KUKA KRL program: MyProgram_153().src

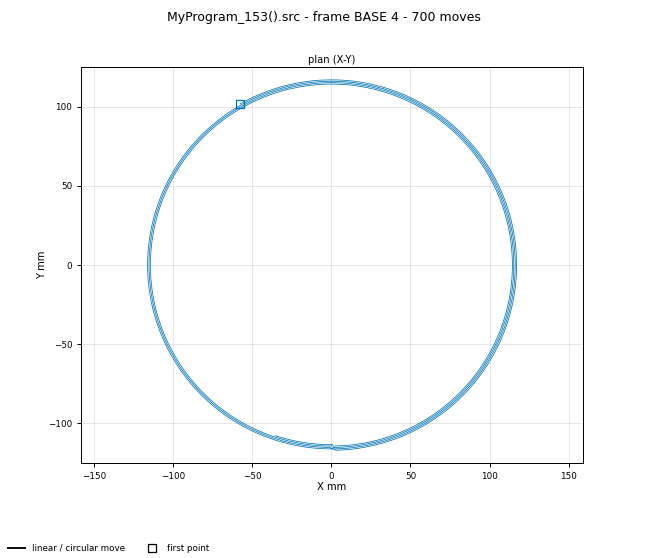
[picture p0: tool path of MyProgram_153().src in frame BASE 4, 700 of 700 moves have a stored position in this frame; points joined in program order, loops and branches not executed]
&ACCESS RVP
&REL 1
&PARAM TEMPLATE = C:\KRC\Roboter\Template\vorgabe
&PARAM EDITMASK = *
DEF MyProgram_153()
; ---- Setting reference (Base) ----
$BASE = BASE_DATA[4]

; --------------------------
; ---- Setting tool (TCP) ----
$TOOL = TOOL_DATA[3]
; --------------------------

$VEL.CP = VEL_APROX_PRINT
Startdeposition()
$VEL.CP = VEL_PRINT
LIN {X -57.7236,Y 101.8964,Z 119,A 114.9153,B 24.9392,C -1.8008,E1 24.9221,E2 331.1013} C_DIS
LIN {X -55.2055,Y 103.2823,Z 119,A 113.5039,B 24.9391,C -1.803,E1 24.9256,E2 332.5114} C_DIS
LIN {X -52.6542,Y 104.606,Z 119,A 112.0926,B 24.9389,C -1.8052,E1 24.9291,E2 333.9216} C_DIS
LIN {X -49.1645,Y 106.2888,Z 119,A 110.1729,B 24.9388,C -1.8071,E1 24.9339,E2 335.8414} C_DIS
LIN {X -46.1406,Y 107.638,Z 119,A 108.5652,B 24.9386,C -1.81,E1 24.938,E2 337.446} C_DIS
LIN {X -43.7577,Y 108.627,Z 119,A 107.2769,B 24.9386,C -1.8107,E1 24.9413,E2 338.7355} C_DIS
LIN {X -40.8035,Y 109.7723,Z 119,A 105.7445,B 24.9384,C -1.8135,E1 24.9453,E2 340.2645} C_DIS
LIN {X -38.3749,Y 110.6432,Z 119,A 104.5039,B 24.9382,C -1.8161,E1 24.9486,E2 341.5015} C_DIS
LIN {X -35.3681,Y 111.6422,Z 119,A 102.9247,B 24.9382,C -1.8167,E1 24.9528,E2 343.0821} C_DIS
LIN {X -32.8997,Y 112.3929,Z 119,A 101.6757,B 24.938,C -1.8187,E1 24.9561,E2 344.3285} C_DIS
LIN {X -30.1315,Y 113.1665,Z 119,A 100.2276,B 24.938,C -1.8184,E1 24.96,E2 345.7796} C_DIS
LIN {X -27.0594,Y 113.9416,Z 119,A 98.6962,B 24.9379,C -1.8206,E1 24.9642,E2 347.3077} C_DIS
LIN {X -24.5424,Y 114.5086,Z 119,A 97.4094,B 24.9379,C -1.8207,E1 24.9677,E2 348.5959} C_DIS
LIN {X -21.7248,Y 115.0764,Z 119,A 96.023,B 24.9377,C -1.8227,E1 24.9715,E2 349.979} C_DIS
LIN {X -18.8941,Y 115.5749,Z 119,A 94.5921,B 24.9377,C -1.8227,E1 24.9754,E2 351.4114} C_DIS
LIN {X -16.1821,Y 115.9853,Z 119,A 93.2548,B 24.9377,C -1.8238,E1 24.9791,E2 352.7472} C_DIS
LIN {X -12.9082,Y 116.397,Z 119,A 91.6544,B 24.9375,C -1.8253,E1 24.9835,E2 354.3452} C_DIS
LIN {X -10.0478,Y 116.6787,Z 119,A 90.2465,B 24.9375,C -1.8259,E1 24.9875,E2 355.7523} C_DIS
LIN {X -7.1813,Y 116.8902,Z 119,A 88.839,B 24.9375,C -1.8265,E1 24.9914,E2 357.159} C_DIS
LIN {X -4.3105,Y 117.0312,Z 119,A 87.4316,B 24.9375,C -1.8269,E1 24.9953,E2 358.5658} C_DIS
LIN {X -1.7313,Y 117.0963,Z 119,A 86.1688,B 24.9375,C -1.8272,E1 24.9988,E2 359.8279} C_DIS
LIN {X 1.4371,Y 117.1018,Z 119,A 84.6179,B 24.9375,C -1.8274,E1 25.0032,E2 361.3782} C_DIS
LIN {X 4.0165,Y 117.0403,Z 119,A 83.3552,B 24.9374,C -1.8276,E1 25.0067,E2 362.6403} C_DIS
LIN {X 7.1813,Y 116.8902,Z 119,A 81.8052,B 24.9374,C -1.8276,E1 25.011,E2 364.1896} C_DIS
LIN {X 10.0478,Y 116.6787,Z 119,A 80.399,B 24.9374,C -1.8275,E1 25.0149,E2 365.5954} C_DIS
LIN {X 12.9082,Y 116.397,Z 119,A 78.9934,B 24.9374,C -1.8273,E1 25.0188,E2 367.0004} C_DIS
LIN {X 15.7608,Y 116.0452,Z 119,A 77.5876,B 24.9374,C -1.827,E1 25.0227,E2 368.4058} C_DIS
LIN {X 18.3132,Y 115.6684,Z 119,A 76.3039,B 24.9375,C -1.8257,E1 25.0263,E2 369.6914} C_DIS
LIN {X 21.1464,Y 115.1841,Z 119,A 74.8988,B 24.9375,C -1.8252,E1 25.0301,E2 371.0961} C_DIS
LIN {X 23.9667,Y 114.6305,Z 119,A 73.4939,B 24.9375,C -1.8247,E1 25.034,E2 372.5007} C_DIS
LIN {X 26.7727,Y 114.0078,Z 119,A 72.1234,B 24.9375,C -1.8255,E1 25.0377,E2 373.8673} C_DIS
LIN {X 29.5625,Y 113.3164,Z 119,A 70.6849,B 24.9377,C -1.8232,E1 25.0416,E2 375.3091} C_DIS
LIN {X 32.3345,Y 112.5568,Z 119,A 69.2808,B 24.9377,C -1.8223,E1 25.0454,E2 376.7129} C_DIS
LIN {X 35.3681,Y 111.6422,Z 119,A 67.7553,B 24.9377,C -1.8223,E1 25.0494,E2 378.236} C_DIS
LIN {X 38.0973,Y 110.7406,Z 119,A 66.3515,B 24.9378,C -1.8211,E1 25.0531,E2 379.6396} C_DIS
LIN {X 40.5271,Y 109.8731,Z 119,A 65.0695,B 24.938,C -1.8191,E1 25.0565,E2 380.9237} C_DIS
LIN {X 43.2113,Y 108.8455,Z 119,A 63.6885,B 24.938,C -1.8188,E1 25.0601,E2 382.3024} C_DIS
LIN {X 45.7716,Y 107.7935,Z 119,A 62.3622,B 24.938,C -1.8186,E1 25.0635,E2 383.626} C_DIS
LIN {X 48.5001,Y 106.5941,Z 119,A 60.8826,B 24.9382,C -1.816,E1 25.0673,E2 385.1081} C_DIS
LIN {X 51.3666,Y 105.2443,Z 119,A 59.3365,B 24.9383,C -1.8142,E1 25.0712,E2 386.6544} C_DIS
LIN {X 53.672,Y 104.0859,Z 119,A 58.0778,B 24.9384,C -1.8128,E1 25.0743,E2 387.913} C_DIS
LIN {X 56.4688,Y 102.5971,Z 119,A 56.5322,B 24.9385,C -1.8108,E1 25.0781,E2 389.4588} C_DIS
LIN {X 58.9697,Y 101.1804,Z 119,A 55.1304,B 24.9387,C -1.809,E1 25.0815,E2 390.8608} C_DIS
LIN {X 61.435,Y 99.7027,Z 119,A 53.7287,B 24.9387,C -1.8071,E1 25.0849,E2 392.2626} C_DIS
LIN {X 63.8633,Y 98.165,Z 119,A 52.3274,B 24.9389,C -1.8051,E1 25.0881,E2 393.6641} C_DIS
LIN {X 67.1917,Y 95.9158,Z 119,A 50.3687,B 24.9391,C -1.8021,E1 25.0927,E2 395.6232} C_DIS
LIN {X 69.5253,Y 94.2379,Z 119,A 48.9459,B 24.9393,C -1.7989,E1 25.0959,E2 397.0486} C_DIS
LIN {X 72.0501,Y 92.3237,Z 119,A 47.424,B 24.9395,C -1.7973,E1 25.0992,E2 398.5686} C_DIS
LIN {X 74.2942,Y 90.5277,Z 119,A 46.023,B 24.9396,C -1.7949,E1 25.1023,E2 399.97} C_DIS
LIN {X 76.1743,Y 88.9491,Z 119,A 44.8121,B 24.9398,C -1.7921,E1 25.1049,E2 401.1827} C_DIS
LIN {X 78.6467,Y 86.7732,Z 119,A 43.2226,B 24.94,C -1.7899,E1 25.1082,E2 402.7713} C_DIS
LIN {X 80.5382,Y 85.0185,Z 119,A 41.9437,B 24.9402,C -1.7865,E1 25.1108,E2 404.0529} C_DIS
LIN {X 82.4233,Y 83.1914,Z 119,A 40.6216,B 24.9405,C -1.782,E1 25.1134,E2 405.3801} C_DIS
LIN {X 84.817,Y 80.7525,Z 119,A 39.0233,B 24.9405,C -1.7817,E1 25.1165,E2 406.9722} C_DIS
LIN {X 86.7732,Y 78.6467,Z 119,A 37.6237,B 24.9407,C -1.7788,E1 25.1192,E2 408.3724} C_DIS
LIN {X 89.4184,Y 75.6234,Z 119,A 35.6681,B 24.941,C -1.7747,E1 25.1227,E2 410.3289} C_DIS
LIN {X 91.2474,Y 73.4062,Z 119,A 34.2691,B 24.9412,C -1.7717,E1 25.1252,E2 411.7284} C_DIS
LIN {X 93.2009,Y 70.9117,Z 119,A 32.7271,B 24.9414,C -1.7683,E1 25.1278,E2 413.2713} C_DIS
LIN {X 95.424,Y 67.8871,Z 119,A 30.862,B 24.9418,C -1.7623,E1 25.1309,E2 415.1414} C_DIS
LIN {X 97.2089,Y 65.3068,Z 119,A 29.3517,B 24.942,C -1.7595,E1 25.1333,E2 416.6509} C_DIS
LIN {X 98.7132,Y 63.0092,Z 119,A 28.0222,B 24.9422,C -1.7567,E1 25.1353,E2 417.9804} C_DIS
LIN {X 100.2963,Y 60.4583,Z 119,A 26.5548,B 24.9424,C -1.7528,E1 25.1374,E2 419.4494} C_DIS
LIN {X 101.8964,Y 57.7236,Z 119,A 25.036,B 24.9426,C -1.75,E1 25.1396,E2 420.967} C_DIS
LIN {X 103.142,Y 55.4641,Z 119,A 23.7809,B 24.9428,C -1.7469,E1 25.1412,E2 422.2228} C_DIS
LIN {X 104.606,Y 52.6542,Z 119,A 22.2401,B 24.9431,C -1.743,E1 25.1432,E2 423.7647} C_DIS
LIN {X 105.7393,Y 50.3364,Z 119,A 20.9634,B 24.9433,C -1.7387,E1 25.1448,E2 425.0446} C_DIS
LIN {X 107.0636,Y 47.458,Z 119,A 19.4448,B 24.9435,C -1.7357,E1 25.1465,E2 426.5621} C_DIS
LIN {X 108.627,Y 43.7577,Z 119,A 17.4694,B 24.9439,C -1.7295,E1 25.1486,E2 428.5412} C_DIS
LIN {X 109.7723,Y 40.8035,Z 119,A 15.9513,B 24.9441,C -1.7264,E1 25.1501,E2 430.0582} C_DIS
LIN {X 110.6432,Y 38.3749,Z 119,A 14.6749,B 24.9444,C -1.722,E1 25.1513,E2 431.3379} C_DIS
LIN {X 111.5517,Y 35.648,Z 119,A 13.2998,B 24.9446,C -1.7192,E1 25.1525,E2 432.7118} C_DIS
LIN {X 112.3929,Y 32.8996,Z 119,A 11.9026,B 24.9449,C -1.7153,E1 25.1536,E2 434.1101} C_DIS
LIN {X 113.1665,Y 30.1315,Z 119,A 10.5341,B 24.945,C -1.7128,E1 25.1546,E2 435.4768} C_DIS
LIN {X 113.8718,Y 27.3452,Z 119,A 9.1088,B 24.9454,C -1.7075,E1 25.1556,E2 436.9064} C_DIS
LIN {X 114.5713,Y 24.2549,Z 119,A 7.5688,B 24.9456,C -1.7031,E1 25.1565,E2 438.4478} C_DIS
LIN {X 115.0764,Y 21.7248,Z 119,A 6.3152,B 24.9459,C -1.6995,E1 25.1572,E2 439.7024} C_DIS
LIN {X 115.5684,Y 18.9331,Z 119,A 4.9099,B 24.9462,C -1.6942,E1 25.1579,E2 441.1119} C_DIS
LIN {X 116.0038,Y 16.0521,Z 119,A 3.5219,B 24.9464,C -1.6915,E1 25.1584,E2 442.4983} C_DIS
LIN {X 116.397,Y 12.9082,Z 119,A 1.9824,B 24.9467,C -1.687,E1 25.1589,E2 444.0393} C_DIS
LIN {X 116.6517,Y 10.3407,Z 119,A 0.7286,B 24.9469,C -1.6833,E1 25.1592,E2 445.2942} C_DIS
LIN {X 116.8902,Y 7.1813,Z 119,A -0.8108,B 24.9472,C -1.6788,E1 25.1595,E2 446.8353} C_DIS
LIN {X 117.0312,Y 4.3105,Z 119,A -2.2075,B 24.9474,C -1.6747,E1 25.1597,E2 448.2333} C_DIS
LIN {X 117.0963,Y 1.7313,Z 119,A -3.497,B 24.9478,C -1.6693,E1 25.1597,E2 449.5278} C_DIS
LIN {X 117.0963,Y -1.7313,Z 119,A -5.014,B 24.9476,C -1.6722,E1 25.1597,E2 451.0289} C_DIS
LIN {X 117.0465,Y -3.8126,Z 119,A -6.1822,B 24.9483,C -1.6618,E1 25.1597,E2 452.2148} C_DIS
LIN {X 116.91,Y -6.8222,Z 119,A -7.6255,B 24.9485,C -1.6584,E1 25.1595,E2 453.6574} C_DIS
LIN {X 116.693,Y -9.8691,Z 119,A -9.1115,B 24.9487,C -1.6539,E1 25.1591,E2 455.1452} C_DIS
LIN {X 116.397,Y -12.9082,Z 119,A -10.586,B 24.949,C -1.6499,E1 25.1587,E2 456.6204} C_DIS
LIN {X 116.0452,Y -15.7608,Z 119,A -11.9826,B 24.9492,C -1.6458,E1 25.1582,E2 458.0185} C_DIS
LIN {X 115.6684,Y -18.3132,Z 119,A -13.2584,B 24.9495,C -1.6411,E1 25.1577,E2 459.2978} C_DIS
LIN {X 115.1321,Y -21.4359,Z 119,A -14.7758,B 24.9497,C -1.6376,E1 25.1569,E2 460.8147} C_DIS
LIN {X 114.6305,Y -23.9667,Z 119,A -16.0514,B 24.95,C -1.6329,E1 25.1562,E2 462.0939} C_DIS
LIN {X 114.0078,Y -26.7727,Z 119,A -17.426,B 24.9502,C -1.6299,E1 25.1554,E2 463.4677} C_DIS
LIN {X 113.3164,Y -29.5625,Z 119,A -18.8446,B 24.9505,C -1.6248,E1 25.1544,E2 464.89} C_DIS
LIN {X 112.2191,Y -33.4857,Z 119,A -20.8654,B 24.951,C -1.6171,E1 25.1528,E2 466.9174} C_DIS
LIN {X 111.2904,Y -36.4555,Z 119,A -22.3142,B 24.951,C -1.6157,E1 25.1516,E2 468.3612} C_DIS
LIN {X 110.4329,Y -38.9742,Z 119,A -23.6361,B 24.9514,C -1.6107,E1 25.1504,E2 469.6876} C_DIS
LIN {X 109.3675,Y -41.8724,Z 119,A -25.108,B 24.9516,C -1.6078,E1 25.1489,E2 471.158} C_DIS
LIN {X 108.1961,Y -44.8163,Z 119,A -26.6478,B 24.9518,C -1.6035,E1 25.1473,E2 472.6996} C_DIS
LIN {X 107.1812,Y -47.1884,Z 119,A -27.9239,B 24.9521,C -1.5989,E1 25.1459,E2 473.9794} C_DIS
LIN {X 105.8667,Y -50.0712,Z 119,A -29.442,B 24.9523,C -1.5957,E1 25.1441,E2 475.4969} C_DIS
LIN {X 104.606,Y -52.6542,Z 119,A -30.8392,B 24.9525,C -1.5919,E1 25.1424,E2 476.8956} C_DIS
LIN {X 103.4194,Y -54.9452,Z 119,A -32.0936,B 24.9527,C -1.5885,E1 25.1408,E2 478.1514} C_DIS
LIN {X 102.0398,Y -57.4667,Z 119,A -33.491,B 24.9529,C -1.5848,E1 25.1389,E2 479.5502} C_DIS
LIN {X 100.5988,Y -59.9536,Z 119,A -34.9105,B 24.9532,C -1.58,E1 25.1368,E2 480.9736} C_DIS
LIN {X 98.9413,Y -62.6539,Z 119,A -36.4291,B 24.9534,C -1.577,E1 25.1346,E2 482.4916} C_DIS
LIN {X 97.3739,Y -65.0632,Z 119,A -37.8269,B 24.9536,C -1.5734,E1 25.1325,E2 483.891} C_DIS
LIN {X 95.9158,Y -67.1917,Z 119,A -39.0816,B 24.9538,C -1.5703,E1 25.1305,E2 485.1469} C_DIS
LIN {X 94.352,Y -69.3694,Z 119,A -40.4109,B 24.9541,C -1.5658,E1 25.1283,E2 486.4804} C_DIS
LIN {X 92.5033,Y -71.8171,Z 119,A -41.8777,B 24.9542,C -1.5633,E1 25.1258,E2 487.9461} C_DIS
LIN {X 90.5277,Y -74.2942,Z 119,A -43.4188,B 24.9544,C -1.5595,E1 25.1231,E2 489.4889} C_DIS
LIN {X 88.868,Y -76.2695,Z 119,A -44.6741,B 24.9546,C -1.5566,E1 25.1208,E2 490.7455} C_DIS
LIN {X 86.7732,Y -78.6467,Z 119,A -46.2156,B 24.9548,C -1.5529,E1 25.1179,E2 492.2887} C_DIS
LIN {X 84.9044,Y -80.6596,Z 119,A -47.557,B 24.955,C -1.5497,E1 25.1154,E2 493.6319} C_DIS
LIN {X 82.8097,Y -82.8097,Z 119,A -49.0132,B 24.9552,C -1.5466,E1 25.1125,E2 495.0892} C_DIS
LIN {X 80.9643,Y -84.6128,Z 119,A -50.2689,B 24.9553,C -1.5439,E1 25.11,E2 496.3461} C_DIS
LIN {X 78.8634,Y -86.5743,Z 119,A -51.668,B 24.9555,C -1.5409,E1 25.1071,E2 497.7467} C_DIS
LIN {X 76.4935,Y -88.6772,Z 119,A -53.2105,B 24.9557,C -1.5376,E1 25.1039,E2 499.2907} C_DIS
LIN {X 74.5204,Y -90.3397,Z 119,A -54.467,B 24.9559,C -1.535,E1 25.1012,E2 500.5485} C_DIS
LIN {X 72.0501,Y -92.3237,Z 119,A -56.0095,B 24.956,C -1.5319,E1 25.0978,E2 502.0925} C_DIS
LIN {X 69.7627,Y -94.0641,Z 119,A -57.4095,B 24.9562,C -1.5292,E1 25.0947,E2 503.4938} C_DIS
LIN {X 67.4332,Y -95.7478,Z 119,A -58.8096,B 24.9563,C -1.5266,E1 25.0915,E2 504.8953} C_DIS
LIN {X 65.3068,Y -97.2089,Z 119,A -60.0666,B 24.9565,C -1.5243,E1 25.0886,E2 506.1534} C_DIS
LIN {X 62.9015,Y -98.7824,Z 119,A -61.4668,B 24.9566,C -1.5218,E1 25.0853,E2 507.555} C_DIS
LIN {X 60.4583,Y -100.2963,Z 119,A -62.8848,B 24.9568,C -1.5186,E1 25.0819,E2 508.9761} C_DIS
LIN {X 57.7236,Y -101.8964,Z 119,A -64.4114,B 24.9568,C -1.5168,E1 25.0782,E2 510.5023} C_DIS
LIN {X 55.2055,Y -103.2823,Z 119,A -65.8123,B 24.957,C -1.5146,E1 25.0748,E2 511.9044} C_DIS
LIN {X 52.884,Y -104.4886,Z 119,A -67.0847,B 24.9571,C -1.5128,E1 25.0716,E2 513.1776} C_DIS
LIN {X 50.3364,Y -105.7393,Z 119,A -68.4714,B 24.9572,C -1.5106,E1 25.0681,E2 514.5657} C_DIS
LIN {X 47.7263,Y -106.9428,Z 119,A -69.8951,B 24.9574,C -1.5076,E1 25.0645,E2 515.993} C_DIS
LIN {X 45.0874,Y -108.0818,Z 119,A -71.2747,B 24.9574,C -1.5068,E1 25.0609,E2 517.3714} C_DIS
LIN {X 42.1475,Y -109.2633,Z 119,A -72.8202,B 24.9576,C -1.5048,E1 25.0569,E2 518.9181} C_DIS
LIN {X 39.4534,Y -110.2648,Z 119,A -74.2224,B 24.9576,C -1.5031,E1 25.0532,E2 520.3214} C_DIS
LIN {X 36.7355,Y -111.1998,Z 119,A -75.6249,B 24.9578,C -1.5015,E1 25.0495,E2 521.725} C_DIS
LIN {X 34.2764,Y -111.9807,Z 119,A -76.8841,B 24.9578,C -1.5001,E1 25.0462,E2 522.9851} C_DIS
LIN {X 31.5179,Y -112.7882,Z 119,A -78.2869,B 24.9579,C -1.4987,E1 25.0424,E2 524.3888} C_DIS
LIN {X 28.4555,Y -113.6009,Z 119,A -79.8337,B 24.958,C -1.4972,E1 25.0382,E2 525.9368} C_DIS
LIN {X 26.1295,Y -114.1564,Z 119,A -81.026,B 24.9581,C -1.4951,E1 25.035,E2 527.1324} C_DIS
LIN {X 22.8471,Y -114.8603,Z 119,A -82.6405,B 24.9581,C -1.4949,E1 25.0306,E2 528.7455} C_DIS
LIN {X 20.311,Y -115.3344,Z 119,A -83.9008,B 24.9581,C -1.494,E1 25.0271,E2 530.0065} C_DIS
LIN {X 17.1837,Y -115.843,Z 119,A -85.4485,B 24.9582,C -1.4929,E1 25.0228,E2 531.5551} C_DIS
LIN {X 14.6273,Y -116.1921,Z 119,A -86.7314,B 24.9583,C -1.4912,E1 25.0193,E2 532.8411} C_DIS
LIN {X 11.7714,Y -116.516,Z 119,A -88.1136,B 24.9583,C -1.4915,E1 25.0154,E2 534.2218} C_DIS
LIN {X 8.9085,Y -116.7698,Z 119,A -89.5405,B 24.9584,C -1.4898,E1 25.0114,E2 535.6518} C_DIS
LIN {X 6.0401,Y -116.9533,Z 119,A -90.9095,B 24.9584,C -1.4909,E1 25.0076,E2 537.0177} C_DIS
LIN {X 2.874,Y -117.0753,Z 119,A -92.4722,B 24.9584,C -1.4898,E1 25.0033,E2 538.5827} C_DIS
LIN {X 2.874,Y -117.0753,Z 119,A -92.4722,B 24.9584,C -1.4898,E1 25.0033,E2 538.5827} C_DIS
Enddeposition()
LIN {X 0.8107,Y -116.2129,Z 119,A -92.8235,B 24.9559,C -1.5347,E1 25.0026,E2 538.8274} C_DIS
Startdeposition()
$VEL.CP = VEL_PRINT
LIN {X 4.253,Y -116.1409,Z 119,A -90.9838,B 24.9555,C -1.5417,E1 25.0078,E2 536.9717} C_DIS
LIN {X 8.3855,Y -115.9152,Z 119,A -89.0694,B 24.9557,C -1.5369,E1 25.0131,E2 535.0695} C_DIS
LIN {X 11.4655,Y -115.6516,Z 119,A -87.6523,B 24.956,C -1.5328,E1 25.017,E2 533.6628} C_DIS
LIN {X 14.4704,Y -115.3134,Z 119,A -85.9882,B 24.9555,C -1.5417,E1 25.0216,E2 531.979} C_DIS
LIN {X 18.8822,Y -114.673,Z 119,A -83.5014,B 24.9546,C -1.5565,E1 25.0286,E2 529.4595} C_DIS
LIN {X 22.2001,Y -114.077,Z 119,A -81.8222,B 24.9545,C -1.5587,E1 25.0332,E2 527.777} C_DIS
LIN {X 25.6561,Y -113.3507,Z 119,A -80.4241,B 24.9553,C -1.5446,E1 25.0369,E2 526.4143} C_DIS
LIN {X 30.8978,Y -112.0359,Z 119,A -77.7136,B 24.955,C -1.5494,E1 25.0443,E2 523.6965} C_DIS
LIN {X 34.2636,Y -111.0512,Z 119,A -76.0256,B 24.955,C -1.5496,E1 25.0488,E2 522.011} C_DIS
LIN {X 37.4676,Y -110.0121,Z 119,A -74.4944,B 24.9552,C -1.5457,E1 25.0528,E2 520.492} C_DIS
LIN {X 40.0272,Y -109.1065,Z 119,A -73.0582,B 24.9549,C -1.552,E1 25.0566,E2 519.0439} C_DIS
LIN {X 44.6117,Y -107.3148,Z 119,A -70.7821,B 24.9551,C -1.5485,E1 25.0625,E2 516.7813} C_DIS
LIN {X 47.9397,Y -105.8687,Z 119,A -68.956,B 24.9548,C -1.5529,E1 25.0671,E2 514.9491} C_DIS
LIN {X 51.1277,Y -104.3676,Z 119,A -66.9334,B 24.9539,C -1.569,E1 25.0723,E2 512.8938} C_DIS
LIN {X 55.4285,Y -102.1471,Z 119,A -64.8466,B 24.9545,C -1.5592,E1 25.0774,E2 510.8361} C_DIS
LIN {X 58.5784,Y -100.376,Z 119,A -63.1081,B 24.9544,C -1.5604,E1 25.0816,E2 509.1} C_DIS
LIN {X 60.8412,Y -99.0203,Z 119,A -61.7959,B 24.9542,C -1.5634,E1 25.0847,E2 507.7848} C_DIS
LIN {X 62.8687,Y -97.744,Z 119,A -60.6023,B 24.954,C -1.5663,E1 25.0876,E2 506.5882} C_DIS
LIN {X 65.3722,Y -96.0879,Z 119,A -59.0534,B 24.9537,C -1.5725,E1 25.0912,E2 505.0298} C_DIS
LIN {X 68.06,Y -94.2054,Z 119,A -57.5231,B 24.9537,C -1.5717,E1 25.0946,E2 503.5066} C_DIS
LIN {X 70.0238,Y -92.7529,Z 119,A -56.3173,B 24.9536,C -1.5744,E1 25.0973,E2 502.2989} C_DIS
LIN {X 72.184,Y -91.0815,Z 119,A -54.9676,B 24.9534,C -1.5775,E1 25.1003,E2 500.9468} C_DIS
LIN {X 74.9817,Y -88.7938,Z 119,A -53.1012,B 24.9529,C -1.5855,E1 25.1043,E2 499.0687} C_DIS
LIN {X 77.5595,Y -86.5499,Z 119,A -51.4398,B 24.9527,C -1.5884,E1 25.1078,E2 497.4072} C_DIS
LIN {X 79.9992,Y -84.3015,Z 119,A -49.914,B 24.9528,C -1.5871,E1 25.1109,E2 495.8907} C_DIS
LIN {X 81.9579,Y -82.3979,Z 119,A -48.4044,B 24.9521,C -1.5981,E1 25.1139,E2 494.3614} C_DIS
LIN {X 84.5156,Y -79.7716,Z 119,A -46.7091,B 24.9521,C -1.5973,E1 25.1172,E2 492.6753} C_DIS
LIN {X 87.0213,Y -77.0329,Z 119,A -44.7713,B 24.9516,C -1.6071,E1 25.1208,E2 490.7229} C_DIS
LIN {X 89.4873,Y -74.1512,Z 119,A -43.0863,B 24.9518,C -1.6033,E1 25.1238,E2 489.0547} C_DIS
LIN {X 91.1471,Y -72.101,Z 119,A -41.76,B 24.9515,C -1.608,E1 25.1262,E2 487.7234} C_DIS
LIN {X 93.2609,Y -69.3475,Z 119,A -40.0948,B 24.9515,C -1.6105,E1 25.129,E2 486.0604} C_DIS
LIN {X 95.3441,Y -66.452,Z 119,A -38.2246,B 24.9508,C -1.6207,E1 25.132,E2 484.175} C_DIS
LIN {X 97.3147,Y -63.5332,Z 119,A -36.3931,B 24.9502,C -1.6302,E1 25.1348,E2 482.3303} C_DIS
LIN {X 100.5499,Y -58.2774,Z 119,A -33.6602,B 24.9506,C -1.6242,E1 25.1388,E2 479.6255} C_DIS
LIN {X 101.9362,Y -55.8173,Z 119,A -32.1145,B 24.9499,C -1.6357,E1 25.1409,E2 478.0608} C_DIS
LIN {X 103.6714,Y -52.524,Z 119,A -29.9709,B 24.9486,C -1.656,E1 25.1436,E2 475.8807} C_DIS
LIN {X 105.143,Y -49.5133,Z 119,A -28.8351,B 24.9498,C -1.6362,E1 25.145,E2 474.7976} C_DIS
LIN {X 106.0516,Y -47.5339,Z 119,A -27.6856,B 24.9494,C -1.6432,E1 25.1463,E2 473.6381} C_DIS
LIN {X 107.4428,Y -44.3021,Z 119,A -26.0414,B 24.9494,C -1.6442,E1 25.1481,E2 472.0004} C_DIS
LIN {X 108.4294,Y -41.8321,Z 119,A -24.6571,B 24.9489,C -1.6518,E1 25.1495,E2 470.606} C_DIS
LIN {X 109.2722,Y -39.5727,Z 119,A -23.4046,B 24.9485,C -1.6586,E1 25.1507,E2 469.3445} C_DIS
LIN {X 110.5377,Y -35.8857,Z 119,A -21.4658,B 24.948,C -1.6655,E1 25.1524,E2 467.4004} C_DIS
LIN {X 111.4364,Y -32.9893,Z 119,A -20.0248,B 24.9479,C -1.6676,E1 25.1536,E2 465.9625} C_DIS
LIN {X 112.4888,Y -29.201,Z 119,A -18.0887,B 24.9475,C -1.6737,E1 25.155,E2 464.0231} C_DIS
LIN {X 113.4181,Y -25.3586,Z 119,A -16.0726,B 24.9469,C -1.6832,E1 25.1563,E2 461.9963} C_DIS
LIN {X 114.2163,Y -21.4768,Z 119,A -14.1057,B 24.9465,C -1.6902,E1 25.1573,E2 460.0245} C_DIS
LIN {X 114.9223,Y -17.3041,Z 119,A -12.1735,B 24.9465,C -1.6896,E1 25.1582,E2 458.1051} C_DIS
LIN {X 115.4268,Y -13.5277,Z 119,A -10.266,B 24.946,C -1.6971,E1 25.1588,E2 456.1911} C_DIS
LIN {X 115.7339,Y -10.5844,Z 119,A -8.8175,B 24.9458,C -1.7014,E1 25.1592,E2 454.7411} C_DIS
LIN {X 116.0065,Y -7.0137,Z 119,A -6.9886,B 24.9452,C -1.7102,E1 25.1596,E2 452.9024} C_DIS
LIN {X 116.1771,Y -3.0757,Z 119,A -5.2194,B 24.9453,C -1.7081,E1 25.1598,E2 451.1484} C_DIS
LIN {X 116.215,Y -0.6787,Z 119,A -4.0416,B 24.9451,C -1.7118,E1 25.1598,E2 449.9689} C_DIS
LIN {X 116.1972,Y 2.1365,Z 119,A -2.5867,B 24.9446,C -1.7196,E1 25.1598,E2 448.5045} C_DIS
LIN {X 116.1033,Y 5.1384,Z 119,A -1.1929,B 24.9446,C -1.7202,E1 25.1596,E2 447.1174} C_DIS
LIN {X 115.9024,Y 8.571,Z 119,A 0.4861,B 24.9442,C -1.7249,E1 25.1593,E2 445.4374} C_DIS
LIN {X 115.6815,Y 11.1514,Z 119,A 1.738,B 24.9441,C -1.7278,E1 25.159,E2 444.186} C_DIS
LIN {X 115.354,Y 14.1499,Z 119,A 3.2576,B 24.9436,C -1.7341,E1 25.1585,E2 442.6604} C_DIS
LIN {X 114.8631,Y 17.6866,Z 119,A 4.9746,B 24.9434,C -1.7377,E1 25.1578,E2 440.9451} C_DIS
LIN {X 114.3714,Y 20.6285,Z 119,A 6.5239,B 24.9429,C -1.7462,E1 25.157,E2 439.385} C_DIS
LIN {X 112.7269,Y 28.2747,Z 119,A 10.9009,B 24.9404,C -1.7832,E1 25.1543,E2 434.9462} C_DIS
LIN {X 111.6203,Y 32.3693,Z 119,A 12.3577,B 24.942,C -1.7592,E1 25.1532,E2 433.5542} C_DIS
LIN {X 110.8416,Y 34.9399,Z 119,A 13.8569,B 24.9412,C -1.7716,E1 25.1519,E2 432.0343} C_DIS
LIN {X 109.644,Y 38.5298,Z 119,A 15.5806,B 24.9412,C -1.7705,E1 25.1504,E2 430.323} C_DIS
LIN {X 108.5425,Y 41.5336,Z 119,A 17.2672,B 24.9406,C -1.7803,E1 25.1487,E2 428.6225} C_DIS
LIN {X 107.103,Y 45.1142,Z 119,A 18.9913,B 24.9408,C -1.7774,E1 25.1469,E2 426.9147} C_DIS
LIN {X 105.6303,Y 48.4665,Z 119,A 20.7455,B 24.9406,C -1.7802,E1 25.1449,E2 425.1635} C_DIS
LIN {X 104.2221,Y 51.4214,Z 119,A 22.4929,B 24.9399,C -1.7912,E1 25.1428,E2 423.3997} C_DIS
LIN {X 102.6122,Y 54.5646,Z 119,A 24.2036,B 24.9396,C -1.7946,E1 25.1405,E2 421.69} C_DIS
LIN {X 100.7406,Y 57.9455,Z 119,A 26.1314,B 24.9392,C -1.8009,E1 25.1379,E2 419.7574} C_DIS
LIN {X 98.8898,Y 61.0535,Z 119,A 27.8696,B 24.939,C -1.8035,E1 25.1354,E2 418.0219} C_DIS
LIN {X 96.4195,Y 64.8826,Z 119,A 30.1003,B 24.9387,C -1.8086,E1 25.132,E2 415.7901} C_DIS
LIN {X 94.333,Y 67.8812,Z 119,A 31.8188,B 24.9387,C -1.8093,E1 25.1292,E2 414.0784} C_DIS
LIN {X 92.5913,Y 70.2388,Z 119,A 33.5412,B 24.9375,C -1.8259,E1 25.1262,E2 412.325} C_DIS
LIN {X 90.3004,Y 73.1586,Z 119,A 35.1466,B 24.9379,C -1.8198,E1 25.1235,E2 410.7416} C_DIS
LIN {X 87.7708,Y 76.1759,Z 119,A 37.1508,B 24.9374,C -1.8273,E1 25.1198,E2 408.7288} C_DIS
LIN {X 84.9502,Y 79.3094,Z 119,A 38.9364,B 24.938,C -1.8183,E1 25.1165,E2 406.9722} C_DIS
LIN {X 83.3255,Y 81.0152,Z 119,A 40.2225,B 24.9375,C -1.8267,E1 25.114,E2 405.672} C_DIS
LIN {X 81.3391,Y 83.0092,Z 119,A 41.9399,B 24.9362,C -1.845,E1 25.1105,E2 403.9184} C_DIS
LIN {X 78.4661,Y 85.7289,Z 119,A 43.5948,B 24.9369,C -1.8353,E1 25.1072,E2 402.2932} C_DIS
LIN {X 75.7231,Y 88.1622,Z 119,A 45.5314,B 24.9362,C -1.8449,E1 25.1031,E2 400.3417} C_DIS
LIN {X 72.1095,Y 91.1404,Z 119,A 47.7484,B 24.9362,C -1.845,E1 25.0983,E2 398.1326} C_DIS
LIN {X 68.9027,Y 93.5888,Z 119,A 50.173,B 24.9345,C -1.8687,E1 25.0927,E2 395.6607} C_DIS
LIN {X 65.6694,Y 95.8867,Z 119,A 51.764,B 24.9355,C -1.8551,E1 25.0892,E2 394.1074} C_DIS
LIN {X 62.1674,Y 98.1939,Z 119,A 53.6266,B 24.9359,C -1.849,E1 25.0849,E2 392.2652} C_DIS
LIN {X 59.197,Y 100.0103,Z 119,A 55.4249,B 24.9355,C -1.8554,E1 25.0805,E2 390.4575} C_DIS
LIN {X 55.9099,Y 101.886,Z 119,A 57.1397,B 24.9358,C -1.8511,E1 25.0764,E2 388.7578} C_DIS
LIN {X 53.8271,Y 103.0007,Z 119,A 58.6381,B 24.9346,C -1.8679,E1 25.0726,E2 387.224} C_DIS
LIN {X 49.8879,Y 104.9657,Z 119,A 60.56,B 24.9352,C -1.8593,E1 25.0678,E2 385.3275} C_DIS
LIN {X 47.3698,Y 106.1255,Z 119,A 61.9307,B 24.9351,C -1.8611,E1 25.0643,E2 383.9561} C_DIS
LIN {X 44.1416,Y 107.5081,Z 119,A 63.7304,B 24.9347,C -1.866,E1 25.0597,E2 382.1488} C_DIS
LIN {X 41.5455,Y 108.538,Z 119,A 64.9955,B 24.935,C -1.8623,E1 25.0564,E2 380.8952} C_DIS
LIN {X 38.3682,Y 109.7007,Z 119,A 66.7171,B 24.9347,C -1.8663,E1 25.0519,E2 379.1678} C_DIS
LIN {X 35.2519,Y 110.7428,Z 119,A 68.2686,B 24.9348,C -1.8645,E1 25.0478,E2 377.6234} C_DIS
LIN {X 32.8299,Y 111.4836,Z 119,A 69.5078,B 24.9348,C -1.865,E1 25.0445,E2 376.3852} C_DIS
LIN {X 29.8854,Y 112.3094,Z 119,A 71.1683,B 24.9342,C -1.8729,E1 25.04,E2 374.7088} C_DIS
LIN {X 25.082,Y 113.4784,Z 119,A 73.4989,B 24.9345,C -1.8694,E1 25.0337,E2 372.3895} C_DIS
LIN {X 21.0146,Y 114.302,Z 119,A 75.3916,B 24.9349,C -1.8635,E1 25.0285,E2 370.5132} C_DIS
LIN {X 18.5873,Y 114.7223,Z 119,A 76.7984,B 24.9343,C -1.8724,E1 25.0246,E2 369.0867} C_DIS
LIN {X 14.5018,Y 115.3093,Z 119,A 78.9421,B 24.9339,C -1.8778,E1 25.0186,E2 366.9321} C_DIS
LIN {X 10.1263,Y 115.7762,Z 119,A 81.1141,B 24.9339,C -1.8781,E1 25.0126,E2 364.7606} C_DIS
LIN {X 5.8984,Y 116.0682,Z 119,A 82.992,B 24.9345,C -1.8688,E1 25.0074,E2 362.9056} C_DIS
LIN {X 3.0351,Y 116.1784,Z 119,A 84.5479,B 24.9341,C -1.875,E1 25.003,E2 361.3354} C_DIS
LIN {X -0.964,Y 116.2131,Z 119,A 86.5503,B 24.9341,C -1.8759,E1 24.9974,E2 359.3307} C_DIS
LIN {X -5.2898,Y 116.0968,Z 119,A 88.5233,B 24.9346,C -1.8683,E1 24.992,E2 357.3757} C_DIS
LIN {X -8.9683,Y 115.8706,Z 119,A 90.1659,B 24.9352,C -1.8599,E1 24.9875,E2 355.7522} C_DIS
LIN {X -11.5624,Y 115.6415,Z 119,A 92.0371,B 24.9334,C -1.8848,E1 24.9821,E2 353.8209} C_DIS
LIN {X -15.3841,Y 115.195,Z 119,A 93.5599,B 24.9346,C -1.8674,E1 24.978,E2 352.3384} C_DIS
LIN {X -18.4835,Y 114.7396,Z 119,A 95.2034,B 24.9344,C -1.8706,E1 24.9734,E2 350.6858} C_DIS
LIN {X -21.8459,Y 114.1452,Z 119,A 96.8124,B 24.9347,C -1.8661,E1 24.969,E2 349.0858} C_DIS
LIN {X -26.8358,Y 113.0782,Z 119,A 99.2894,B 24.935,C -1.8621,E1 24.9623,E2 346.6151} C_DIS
LIN {X -29.5914,Y 112.3885,Z 119,A 100.8887,B 24.9345,C -1.8693,E1 24.9579,E2 344.9965} C_DIS
LIN {X -33.0793,Y 111.4097,Z 119,A 102.5685,B 24.935,C -1.8628,E1 24.9534,E2 343.3294} C_DIS
LIN {X -36.8914,Y 110.2063,Z 119,A 104.5056,B 24.9352,C -1.859,E1 24.9483,E2 341.3978} C_DIS
LIN {X -40.0732,Y 109.0897,Z 119,A 106.4101,B 24.9346,C -1.8672,E1 24.9433,E2 339.47} C_DIS
LIN {X -44.3562,Y 107.4208,Z 119,A 108.6478,B 24.935,C -1.8628,E1 24.9375,E2 337.2377} C_DIS
LIN {X -48.1201,Y 105.7874,Z 119,A 110.3506,B 24.9361,C -1.8462,E1 24.9332,E2 335.5704} C_DIS
LIN {X -51.142,Y 104.3605,Z 119,A 112.0013,B 24.9363,C -1.8437,E1 24.9291,E2 333.9214} C_DIS
LIN {X -54.9067,Y 102.4301,Z 119,A 114.3426,B 24.9358,C -1.851,E1 24.9232,E2 331.5564} C_DIS
LIN {X -58.4929,Y 100.4261,Z 119,A 116.2056,B 24.9365,C -1.8405,E1 24.9187,E2 329.7127} C_DIS
LIN {X -62.111,Y 98.2292,Z 119,A 118.473,B 24.9362,C -1.8442,E1 24.9133,E2 327.4295} C_DIS
LIN {X -65.3177,Y 96.1248,Z 119,A 120.2915,B 24.9367,C -1.8375,E1 24.9091,E2 325.621} C_DIS
LIN {X -67.8817,Y 94.3326,Z 119,A 121.9222,B 24.9367,C -1.838,E1 24.9054,E2 323.9833} C_DIS
LIN {X -70.8859,Y 92.0953,Z 119,A 123.6884,B 24.9372,C -1.8307,E1 24.9015,E2 322.2282} C_DIS
LIN {X -73.2399,Y 90.2346,Z 119,A 125.0905,B 24.9376,C -1.8243,E1 24.8985,E2 320.8362} C_DIS
LIN {X -75.9097,Y 88.0033,Z 119,A 126.8195,B 24.9378,C -1.8209,E1 24.8948,E2 319.1085} C_DIS
LIN {X -78.6596,Y 85.5513,Z 119,A 128.646,B 24.9381,C -1.8172,E1 24.891,E2 317.2835} C_DIS
LIN {X -81.2378,Y 83.1092,Z 119,A 130.3589,B 24.9385,C -1.8114,E1 24.8875,E2 315.5774} C_DIS
LIN {X -83.0787,Y 81.2687,Z 119,A 131.8668,B 24.9381,C -1.8175,E1 24.8846,E2 314.0483} C_DIS
LIN {X -85.5625,Y 78.6474,Z 119,A 133.5682,B 24.9386,C -1.8098,E1 24.8813,E2 312.3579} C_DIS
LIN {X -87.7097,Y 76.2459,Z 119,A 135.1898,B 24.9388,C -1.8071,E1 24.8783,E2 310.7354} C_DIS
LIN {X -89.7416,Y 73.8452,Z 119,A 136.649,B 24.9393,C -1.7992,E1 24.8758,E2 309.2883} C_DIS
LIN {X -92.2553,Y 70.6783,Z 119,A 139.0237,B 24.9386,C -1.8097,E1 24.8716,E2 306.8775} C_DIS
LIN {X -94.1803,Y 68.0948,Z 119,A 140.2409,B 24.94,C -1.7899,E1 24.8697,E2 305.7014} C_DIS
LIN {X -96.5543,Y 64.6835,Z 119,A 142.3074,B 24.9403,C -1.7849,E1 24.8664,E2 303.6366} C_DIS
LIN {X -98.1496,Y 62.2368,Z 119,A 143.9112,B 24.9401,C -1.7876,E1 24.864,E2 302.0183} C_DIS
LIN {X -101.0398,Y 57.4248,Z 119,A 146.7142,B 24.9405,C -1.781,E1 24.86,E2 299.2165} C_DIS
LIN {X -103.1496,Y 53.5443,Z 119,A 148.7319,B 24.9414,C -1.768,E1 24.8574,E2 297.2192} C_DIS
LIN {X -105.6546,Y 48.4133,Z 119,A 151.7085,B 24.9415,C -1.7661,E1 24.8538,E2 294.231} C_DIS
LIN {X -107.0769,Y 45.1762,Z 119,A 153.3993,B 24.942,C -1.7586,E1 24.8519,E2 292.5486} C_DIS
LIN {X -108.4463,Y 41.7876,Z 119,A 155.3086,B 24.9421,C -1.7574,E1 24.85,E2 290.6315} C_DIS
LIN {X -109.702,Y 38.3645,Z 119,A 157.1902,B 24.9423,C -1.7552,E1 24.8482,E2 288.7444} C_DIS
LIN {X -110.8505,Y 34.9111,Z 119,A 158.9065,B 24.9428,C -1.7463,E1 24.8468,E2 287.0394} C_DIS
LIN {X -111.9422,Y 31.2331,Z 119,A 161.1958,B 24.9422,C -1.7566,E1 24.845,E2 284.7123} C_DIS
LIN {X -112.8969,Y 27.5798,Z 119,A 163.0137,B 24.9427,C -1.7489,E1 24.8438,E2 282.9022} C_DIS
LIN {X -113.7062,Y 24.0305,Z 119,A 164.2799,B 24.9445,C -1.7214,E1 24.8431,E2 281.694} C_DIS
LIN {X -114.2849,Y 21.1092,Z 119,A 166.8355,B 24.9419,C -1.7614,E1 24.8418,E2 279.028} C_DIS
LIN {X -115.2127,Y 15.2474,Z 119,A 169.8918,B 24.9421,C -1.7573,E1 24.8406,E2 275.9631} C_DIS
LIN {X -115.8834,Y 8.8091,Z 119,A 172.0075,B 24.9457,C -1.7025,E1 24.8402,E2 273.9655} C_DIS
LIN {X -116.1368,Y 4.3589,Z 119,A 174.3557,B 24.9457,C -1.7015,E1 24.8399,E2 271.6056} C_DIS
LIN {X -116.2092,Y 1.4833,Z 119,A 175.827,B 24.9459,C -1.6991,E1 24.8398,E2 270.1312} C_DIS
LIN {X -116.1936,Y -2.3298,Z 119,A 177.5489,B 24.9467,C -1.6865,E1 24.8398,E2 268.4288} C_DIS
LIN {X -115.998,Y -7.1486,Z 119,A -179.5691,B 24.9459,C -1.6995,E1 24.8403,E2 265.4985} C_DIS
LIN {X -115.7111,Y -10.8307,Z 119,A -178.2347,B 24.9475,C -1.6737,E1 24.8406,E2 264.2178} C_DIS
LIN {X -115.3159,Y -14.4508,Z 119,A -176.3106,B 24.9475,C -1.6732,E1 24.8412,E2 262.2834} C_DIS
LIN {X -114.44,Y -20.2471,Z 119,A -173.6291,B 24.9486,C -1.6554,E1 24.8424,E2 259.6282} C_DIS
LIN {X -113.8399,Y -23.3844,Z 119,A -171.9242,B 24.9486,C -1.6558,E1 24.8433,E2 257.9123} C_DIS
LIN {X -113.1293,Y -26.6144,Z 119,A -170.1397,B 24.9486,C -1.657,E1 24.8444,E2 256.1144} C_DIS
LIN {X -112.1726,Y -30.3918,Z 119,A -168.3018,B 24.9491,C -1.6477,E1 24.8457,E2 254.288} C_DIS
LIN {X -111.2863,Y -33.4951,Z 119,A -166.8233,B 24.9497,C -1.6382,E1 24.8469,E2 252.8238} C_DIS
LIN {X -110.5688,Y -35.7896,Z 119,A -165.4975,B 24.9496,C -1.6404,E1 24.848,E2 251.4851} C_DIS
LIN {X -108.149,Y -42.5458,Z 119,A -162.0073,B 24.9503,C -1.6278,E1 24.8514,E2 248.0051} C_DIS
LIN {X -106.2557,Y -47.0803,Z 119,A -159.5937,B 24.9508,C -1.6203,E1 24.854,E2 245.5959} C_DIS
LIN {X -104.5975,Y -50.6541,Z 119,A -157.6252,B 24.9511,C -1.6159,E1 24.8563,E2 243.6273} C_DIS
LIN {X -103.404,Y -53.0471,Z 119,A -156.2428,B 24.9511,C -1.6149,E1 24.8581,E2 242.2399} C_DIS
LIN {X -101.4489,Y -56.6963,Z 119,A -154.1417,B 24.9513,C -1.6118,E1 24.8609,E2 240.1351} C_DIS
LIN {X -99.8492,Y -59.4696,Z 119,A -152.683,B 24.9519,C -1.6025,E1 24.863,E2 238.6909} C_DIS
LIN {X -98.066,Y -62.3671,Z 119,A -150.9229,B 24.9519,C -1.6015,E1 24.8656,E2 236.9242} C_DIS
LIN {X -96.2075,Y -65.1956,Z 119,A -149.2443,B 24.9522,C -1.5977,E1 24.8682,E2 235.2464} C_DIS
LIN {X -94.4799,Y -67.6753,Z 119,A -147.2054,B 24.951,C -1.617,E1 24.8716,E2 233.1515} C_DIS
LIN {X -92.0441,Y -70.9523,Z 119,A -145.2431,B 24.9514,C -1.6099,E1 24.8749,E2 231.1967} C_DIS
LIN {X -89.6369,Y -73.9712,Z 119,A -144.0076,B 24.9534,C -1.5772,E1 24.877,E2 230.0333} C_DIS
LIN {X -86.9034,Y -77.1646,Z 119,A -141.6452,B 24.953,C -1.5846,E1 24.8813,E2 227.6426} C_DIS
LIN {X -84.2445,Y -80.0599,Z 119,A -139.8363,B 24.9535,C -1.5748,E1 24.8848,E2 225.8491} C_DIS
LIN {X -80.6144,Y -83.7118,Z 119,A -136.7963,B 24.9526,C -1.5908,E1 24.8909,E2 222.7585} C_DIS
LIN {X -77.918,Y -86.2289,Z 119,A -135.001,B 24.9529,C -1.5861,E1 24.8946,E2 220.9671} C_DIS
LIN {X -75.3725,Y -88.461,Z 119,A -133.6679,B 24.9539,C -1.5685,E1 24.8974,E2 219.6707} C_DIS
LIN {X -72.5782,Y -90.77,Z 119,A -132.0125,B 24.9544,C -1.5595,E1 24.9009,E2 218.0305} C_DIS
LIN {X -70.536,Y -92.365,Z 119,A -130.7035,B 24.9544,C -1.5585,E1 24.9038,E2 216.7189} C_DIS
LIN {X -68.3476,Y -93.9952,Z 119,A -129.3296,B 24.9546,C -1.5574,E1 24.9069,E2 215.3428} C_DIS
LIN {X -66.2084,Y -95.5135,Z 119,A -127.9849,B 24.9546,C -1.5574,E1 24.91,E2 213.9934} C_DIS
LIN {X -62.7133,Y -97.8437,Z 119,A -125.8454,B 24.9546,C -1.5571,E1 24.915,E2 211.8478} C_DIS
LIN {X -59.5697,Y -99.7901,Z 119,A -124.016,B 24.9547,C -1.5547,E1 24.9194,E2 210.0186} C_DIS
LIN {X -56.5302,Y -101.5416,Z 119,A -122.0317,B 24.9542,C -1.5633,E1 24.9243,E2 208.0079} C_DIS
LIN {X -53.6954,Y -103.07,Z 119,A -120.7873,B 24.9552,C -1.5463,E1 24.9273,E2 206.8005} C_DIS
LIN {X -50.6615,Y -104.5939,Z 119,A -119.036,B 24.9552,C -1.5476,E1 24.9317,E2 205.0416} C_DIS
LIN {X -47.3073,Y -106.1537,Z 119,A -117.138,B 24.9551,C -1.5488,E1 24.9365,E2 203.1362} C_DIS
LIN {X -44.4803,Y -107.3701,Z 119,A -115.7966,B 24.9556,C -1.5395,E1 24.9399,E2 201.8137} C_DIS
LIN {X -42.0737,Y -108.3345,Z 119,A -114.3631,B 24.9553,C -1.545,E1 24.9437,E2 200.364} C_DIS
LIN {X -38.2181,Y -109.7534,Z 119,A -112.4548,B 24.9557,C -1.5381,E1 24.9487,E2 198.4683} C_DIS
LIN {X -34.5865,Y -110.9511,Z 119,A -110.5279,B 24.9557,C -1.5385,E1 24.9538,E2 196.537} C_DIS
LIN {X -31.2531,Y -111.9365,Z 119,A -108.5875,B 24.9551,C -1.5473,E1 24.9591,E2 194.5725} C_DIS
LIN {X -26.6191,Y -113.1282,Z 119,A -106.2804,B 24.9554,C -1.5437,E1 24.9653,E2 192.2708} C_DIS
LIN {X -23.3044,Y -113.8563,Z 119,A -104.7345,B 24.9557,C -1.5373,E1 24.9695,E2 190.7381} C_DIS
LIN {X -19.1455,Y -114.629,Z 119,A -102.728,B 24.956,C -1.5331,E1 24.975,E2 188.7396} C_DIS
LIN {X -16.3202,Y -115.0652,Z 119,A -101.2754,B 24.9559,C -1.5347,E1 24.979,E2 187.282} C_DIS
LIN {X -13.3282,Y -115.4502,Z 119,A -99.8677,B 24.9561,C -1.5309,E1 24.9829,E2 185.8824} C_DIS
LIN {X -9.9444,Y -115.7926,Z 119,A -98.1199,B 24.9559,C -1.5339,E1 24.9878,E2 184.1265} C_DIS
LIN {X -6.2356,Y -116.0496,Z 119,A -96.1919,B 24.9557,C -1.5383,E1 24.9932,E2 182.1876} C_DIS
LIN {X -2.4218,Y -116.1919,Z 119,A -94.382,B 24.9558,C -1.5353,E1 24.9982,E2 180.3845} C_DIS
LIN {X 0.8107,Y -116.2129,Z 119,A -92.8222,B 24.9559,C -1.5342,E1 25.0026,E2 178.8274} C_DIS
Enddeposition()
LIN {X 0.8107,Y -116.2129,Z 119,A -92.8222,B 24.9559,C -1.5342,E1 25.0026,E2 178.8274} C_DIS
Startdeposition()
$VEL.CP = VEL_PRINT
LIN {X -0.9486,Y -115.3216,Z 119,A -94.4449,B 24.9569,C -1.5162,E1 24.9979,E2 180.4926} C_DIS
LIN {X -5.285,Y -115.2046,Z 119,A -96.8248,B 24.9575,C -1.5062,E1 24.9912,E2 182.8968} C_DIS
LIN {X -9.5465,Y -114.93,Z 119,A -98.8545,B 24.9573,C -1.5102,E1 24.9856,E2 184.9178} C_DIS
LIN {X -12.8632,Y -114.607,Z 119,A -100.4098,B 24.957,C -1.5147,E1 24.9813,E2 186.4633} C_DIS
LIN {X -16.5728,Y -114.1288,Z 119,A -102.5307,B 24.9576,C -1.5037,E1 24.9754,E2 188.6118} C_DIS
LIN {X -21.2444,Y -113.3531,Z 119,A -104.5537,B 24.9568,C -1.5188,E1 24.9699,E2 190.6012} C_DIS
LIN {X -26.5055,Y -112.2394,Z 119,A -107.8525,B 24.9582,C -1.4931,E1 24.9607,E2 193.965} C_DIS
LIN {X -30.4948,Y -111.2213,Z 119,A -109.4265,B 24.957,C -1.5146,E1 24.9566,E2 195.4906} C_DIS
LIN {X -33.8365,Y -110.2502,Z 119,A -111.0681,B 24.9567,C -1.5195,E1 24.9522,E2 197.1231} C_DIS
LIN {X -36.8519,Y -109.2788,Z 119,A -112.6395,B 24.9567,C -1.5209,E1 24.9481,E2 198.6942} C_DIS
LIN {X -40.4234,Y -108.0096,Z 119,A -114.6956,B 24.957,C -1.5152,E1 24.9426,E2 200.7679} C_DIS
LIN {X -44.5443,Y -106.3757,Z 119,A -117.2345,B 24.9577,C -1.5033,E1 24.936,E2 203.3409} C_DIS
LIN {X -48.129,Y -104.8039,Z 119,A -118.5846,B 24.9561,C -1.5306,E1 24.9327,E2 204.6295} C_DIS
LIN {X -55.0988,Y -101.3117,Z 119,A -122.589,B 24.9561,C -1.5299,E1 24.9227,E2 208.6463} C_DIS
LIN {X -58.4482,Y -99.4173,Z 119,A -124.857,B 24.9568,C -1.5177,E1 24.9172,E2 210.95} C_DIS
LIN {X -61.23,Y -97.7283,Z 119,A -126.0795,B 24.9558,C -1.5367,E1 24.9143,E2 212.1312} C_DIS
LIN {X -64.3298,Y -95.717,Z 119,A -127.9024,B 24.9556,C -1.5401,E1 24.9101,E2 213.9519} C_DIS
LIN {X -67.3988,Y -93.582,Z 119,A -129.9022,B 24.9557,C -1.5373,E1 24.9055,E2 215.9652} C_DIS
LIN {X -70.1602,Y -91.529,Z 119,A -131.5967,B 24.9555,C -1.541,E1 24.9017,E2 217.6571} C_DIS
LIN {X -73.2087,Y -89.1113,Z 119,A -133.3966,B 24.955,C -1.5501,E1 24.8979,E2 219.442} C_DIS
LIN {X -75.491,Y -87.1852,Z 119,A -135.0285,B 24.9552,C -1.5468,E1 24.8944,E2 221.088} C_DIS
LIN {X -78.0759,Y -84.8769,Z 119,A -136.7955,B 24.9551,C -1.5485,E1 24.8907,E2 222.8583} C_DIS
LIN {X -82.6589,Y -80.4221,Z 119,A -139.9937,B 24.9547,C -1.5543,E1 24.8844,E2 226.0562} C_DIS
LIN {X -85.4034,Y -77.5021,Z 119,A -141.8322,B 24.9541,C -1.565,E1 24.8809,E2 227.8772} C_DIS
LIN {X -87.2621,Y -75.4028,Z 119,A -143.1983,B 24.9539,C -1.5693,E1 24.8784,E2 229.2393} C_DIS
LIN {X -89.0133,Y -73.3266,Z 119,A -144.5666,B 24.9537,C -1.5717,E1 24.8759,E2 230.6082} C_DIS
LIN {X -91.12,Y -70.6899,Z 119,A -146.8711,B 24.955,C -1.5502,E1 24.8719,E2 232.9747} C_DIS
LIN {X -93.582,Y -67.3988,Z 119,A -148.3875,B 24.9534,C -1.5766,E1 24.8695,E2 234.4355} C_DIS
LIN {X -95.5965,Y -64.5078,Z 119,A -150.0346,B 24.9529,C -1.5853,E1 24.8669,E2 236.07} C_DIS
LIN {X -97.9481,Y -60.8782,Z 119,A -152.3796,B 24.9531,C -1.583,E1 24.8633,E2 238.4326} C_DIS
LIN {X -100.0755,Y -57.3136,Z 119,A -154.3529,B 24.9525,C -1.5921,E1 24.8606,E2 240.3942} C_DIS
LIN {X -102.4025,Y -53.0477,Z 119,A -156.9072,B 24.9525,C -1.5931,E1 24.8572,E2 242.9598} C_DIS
LIN {X -103.9507,Y -49.9417,Z 119,A -158.5364,B 24.9519,C -1.6018,E1 24.8552,E2 244.577} C_DIS
LIN {X -105.327,Y -46.9718,Z 119,A -160.312,B 24.952,C -1.6005,E1 24.8531,E2 246.3656} C_DIS
LIN {X -106.8443,Y -43.4075,Z 119,A -162.0985,B 24.9513,C -1.6117,E1 24.8512,E2 248.1353} C_DIS
LIN {X -109.0798,Y -37.4422,Z 119,A -165.5178,B 24.9513,C -1.6108,E1 24.8479,E2 251.5759} C_DIS
LIN {X -110.5008,Y -33.0082,Z 119,A -167.5773,B 24.9503,C -1.6281,E1 24.8463,E2 253.6061} C_DIS
LIN {X -111.3725,Y -29.9349,Z 119,A -169.2836,B 24.9503,C -1.6281,E1 24.845,E2 255.3222} C_DIS
LIN {X -112.3536,Y -26.0115,Z 119,A -171.2728,B 24.9499,C -1.6352,E1 24.8437,E2 257.3061} C_DIS
LIN {X -113.1248,Y -22.4299,Z 119,A -173.1447,B 24.9497,C -1.6388,E1 24.8426,E2 259.1804} C_DIS
LIN {X -114.204,Y -16.0437,Z 119,A -176.4219,B 24.9492,C -1.6467,E1 24.8412,E2 262.4584} C_DIS
LIN {X -115.0016,Y -8.6513,Z 119,A 179.0233,B 24.9505,C -1.6246,E1 24.84,E2 267.0932} C_DIS
LIN {X -115.2916,Y -2.8656,Z 119,A 177.1877,B 24.9474,C -1.6751,E1 24.8398,E2 268.8194} C_DIS
LIN {X -115.291,Y 2.8863,Z 119,A 173.4799,B 24.9489,C -1.6507,E1 24.84,E2 272.6077} C_DIS
LIN {X -115.0786,Y 7.5425,Z 119,A 171.8478,B 24.9468,C -1.6853,E1 24.8402,E2 274.1673} C_DIS
LIN {X -114.3717,Y 14.7995,Z 119,A 168.5665,B 24.9452,C -1.7107,E1 24.8411,E2 277.4076} C_DIS
LIN {X -113.5546,Y 20.1334,Z 119,A 165.4955,B 24.9456,C -1.7037,E1 24.8425,E2 280.5135} C_DIS
LIN {X -112.8446,Y 23.7992,Z 119,A 163.2891,B 24.9461,C -1.6958,E1 24.8437,E2 282.7519} C_DIS
LIN {X -111.6784,Y 28.7724,Z 119,A 160.9268,B 24.9451,C -1.7109,E1 24.8453,E2 285.092} C_DIS
LIN {X -110.5181,Y 32.9496,Z 119,A 158.8591,B 24.9445,C -1.7212,E1 24.8469,E2 287.1471} C_DIS
LIN {X -108.1471,Y 40.0556,Z 119,A 155.106,B 24.9438,C -1.7316,E1 24.8503,E2 290.8969} C_DIS
LIN {X -107.0907,Y 42.8015,Z 119,A 153.7533,B 24.9432,C -1.7404,E1 24.8516,E2 292.236} C_DIS
LIN {X -105.0177,Y 47.6581,Z 119,A 150.9419,B 24.9432,C -1.741,E1 24.8548,E2 295.0616} C_DIS
LIN {X -103.0133,Y 51.8525,Z 119,A 148.6239,B 24.9428,C -1.7475,E1 24.8576,E2 297.3765} C_DIS
LIN {X -100.9556,Y 55.751,Z 119,A 146.4628,B 24.9423,C -1.7552,E1 24.8605,E2 299.5307} C_DIS
LIN {X -96.506,Y 63.1401,Z 119,A 141.6314,B 24.9429,C -1.7458,E1 24.8676,E2 304.4093} C_DIS
LIN {X -94.1778,Y 66.5615,Z 119,A 139.7473,B 24.9421,C -1.7583,E1 24.8706,E2 306.2728} C_DIS
LIN {X -92.1862,Y 69.2937,Z 119,A 138.0692,B 24.9418,C -1.7629,E1 24.8734,E2 307.9479} C_DIS
LIN {X -90.078,Y 72.0159,Z 119,A 136.776,B 24.9403,C -1.7842,E1 24.8756,E2 309.1965} C_DIS
LIN {X -88.0338,Y 74.4991,Z 119,A 135.1336,B 24.9402,C -1.7866,E1 24.8785,E2 310.8407} C_DIS
LIN {X -86.0036,Y 76.833,Z 119,A 133.3457,B 24.9406,C -1.7805,E1 24.8819,E2 312.6512} C_DIS
LIN {X -82.4873,Y 80.5987,Z 119,A 130.9776,B 24.9396,C -1.7945,E1 24.8864,E2 314.9962} C_DIS
LIN {X -80.0253,Y 83.0414,Z 119,A 129.2742,B 24.9393,C -1.7995,E1 24.8898,E2 316.6947} C_DIS
LIN {X -77.266,Y 85.616,Z 119,A 127.2354,B 24.9395,C -1.7973,E1 24.894,E2 318.7472} C_DIS
LIN {X -73.4958,Y 88.8727,Z 119,A 124.8111,B 24.9389,C -1.8049,E1 24.8992,E2 321.1626} C_DIS
LIN {X -70.3408,Y 91.3898,Z 119,A 122.8757,B 24.9384,C -1.8121,E1 24.9034,E2 323.0881} C_DIS
LIN {X -67.5874,Y 93.4468,Z 119,A 120.9036,B 24.9389,C -1.8049,E1 24.9079,E2 325.0845} C_DIS
LIN {X -62.4985,Y 96.9222,Z 119,A 118.0844,B 24.9379,C -1.8208,E1 24.9144,E2 327.875} C_DIS
LIN {X -59.552,Y 98.7605,Z 119,A 116.3042,B 24.9378,C -1.8218,E1 24.9186,E2 329.6585} C_DIS
LIN {X -57.0625,Y 100.2198,Z 119,A 114.9817,B 24.9373,C -1.8289,E1 24.9218,E2 330.9678} C_DIS
LIN {X -52.6064,Y 102.628,Z 119,A 112.4265,B 24.9371,C -1.8316,E1 24.9281,E2 333.5238} C_DIS
LIN {X -46.3765,Y 105.5899,Z 119,A 108.887,B 24.9371,C -1.8323,E1 24.9371,E2 337.0706} C_DIS
LIN {X -39.6192,Y 108.3062,Z 119,A 105.2767,B 24.9367,C -1.8376,E1 24.9464,E2 340.6762} C_DIS
LIN {X -35.9141,Y 109.5914,Z 119,A 103.3316,B 24.9365,C -1.8401,E1 24.9516,E2 342.6189} C_DIS
LIN {X -33.3941,Y 110.3863,Z 119,A 101.8264,B 24.937,C -1.8335,E1 24.9556,E2 344.1424} C_DIS
LIN {X -29.1113,Y 111.5913,Z 119,A 99.8423,B 24.9362,C -1.8453,E1 24.9609,E2 346.1014} C_DIS
LIN {X -23.2506,Y 112.9572,Z 119,A 96.3696,B 24.9374,C -1.8277,E1 24.9705,E2 349.6202} C_DIS
LIN {X -19.4989,Y 113.6659,Z 119,A 94.9258,B 24.936,C -1.8482,E1 24.9743,E2 351.0169} C_DIS
LIN {X -11.9404,Y 114.7055,Z 119,A 91.2748,B 24.9354,C -1.8564,E1 24.9844,E2 354.651} C_DIS
LIN {X -6.1445,Y 115.1617,Z 119,A 88.2751,B 24.9356,C -1.8529,E1 24.9928,E2 357.6604} C_DIS
LIN {X -2.4166,Y 115.3003,Z 119,A 86.3501,B 24.9358,C -1.8504,E1 24.9982,E2 359.5915} C_DIS
LIN {X 1.7405,Y 115.3128,Z 119,A 83.9539,B 24.9368,C -1.8366,E1 25.0049,E2 362.0203} C_DIS
LIN {X 5.0476,Y 115.2148,Z 119,A 82.6595,B 24.9357,C -1.8517,E1 25.0085,E2 363.2786} C_DIS
LIN {X 9.0021,Y 114.9735,Z 119,A 80.7513,B 24.9356,C -1.8542,E1 25.0138,E2 365.1799} C_DIS
LIN {X 13.2272,Y 114.5644,Z 119,A 78.1864,B 24.9369,C -1.8343,E1 25.021,E2 367.7903} C_DIS
LIN {X 16.8573,Y 114.0884,Z 119,A 76.7179,B 24.9359,C -1.8489,E1 25.025,E2 369.223} C_DIS
LIN {X 21.4847,Y 113.3068,Z 119,A 74.4369,B 24.9359,C -1.8502,E1 25.0312,E2 371.4982} C_DIS
LIN {X 23.9903,Y 112.804,Z 119,A 72.9119,B 24.9366,C -1.8385,E1 25.0355,E2 373.0491} C_DIS
LIN {X 28.3216,Y 111.7943,Z 119,A 70.9359,B 24.936,C -1.8474,E1 25.0408,E2 375.0012} C_DIS
LIN {X 31.8818,Y 110.8317,Z 119,A 69.0736,B 24.9362,C -1.8448,E1 25.0458,E2 376.8666} C_DIS
LIN {X 35.2204,Y 109.8159,Z 119,A 67.3806,B 24.9362,C -1.8452,E1 25.0503,E2 378.5554} C_DIS
LIN {X 37.9943,Y 108.887,Z 119,A 65.8879,B 24.9364,C -1.8422,E1 25.0542,E2 380.0523} C_DIS
LIN {X 41.6378,Y 107.5478,Z 119,A 63.5768,B 24.9377,C -1.8235,E1 25.0604,E2 382.4026} C_DIS
LIN {X 45.0948,Y 106.1437,Z 119,A 62.1491,B 24.9365,C -1.8403,E1 25.0639,E2 383.7873} C_DIS
LIN {X 47.6069,Y 105.0408,Z 119,A 60.0427,B 24.9389,C -1.806,E1 25.0695,E2 385.9695} C_DIS
LIN {X 52.3165,Y 102.7761,Z 119,A 58.2042,B 24.9368,C -1.8361,E1 25.0739,E2 387.7319} C_DIS
LIN {X 55.0908,Y 101.316,Z 119,A 56.3607,B 24.9378,C -1.8212,E1 25.0785,E2 389.6052} C_DIS
LIN {X 57.9496,Y 99.71,Z 119,A 55.1343,B 24.9368,C -1.8368,E1 25.0813,E2 390.7911} C_DIS
LIN {X 60.6817,Y 98.0708,Z 119,A 53.4486,B 24.9372,C -1.8298,E1 25.0854,E2 392.4881} C_DIS
LIN {X 62.9331,Y 96.6425,Z 119,A 52.0208,B 24.9377,C -1.823,E1 25.0888,E2 393.9273} C_DIS
LIN {X 66.2927,Y 94.3691,Z 119,A 49.9748,B 24.938,C -1.8183,E1 25.0935,E2 395.9776} C_DIS
LIN {X 69.8307,Y 91.7828,Z 119,A 47.8982,B 24.938,C -1.8189,E1 25.0981,E2 398.0452} C_DIS
LIN {X 74.5812,Y 87.9639,Z 119,A 44.9937,B 24.938,C -1.8187,E1 25.1044,E2 400.939} C_DIS
LIN {X 80.3111,Y 82.7659,Z 119,A 41.1632,B 24.9385,C -1.8114,E1 25.1122,E2 404.7714} C_DIS
LIN {X 83.0341,Y 80.0329,Z 119,A 39.3502,B 24.9385,C -1.812,E1 25.1158,E2 406.5752} C_DIS
LIN {X 86.4561,Y 76.3258,Z 119,A 36.6879,B 24.9393,C -1.7991,E1 25.1208,E2 409.2561} C_DIS
LIN {X 88.4896,Y 73.9568,Z 119,A 34.5901,B 24.9412,C -1.7706,E1 25.1247,E2 411.4116} C_DIS
LIN {X 91.2639,Y 70.5042,Z 119,A 33.0427,B 24.9396,C -1.795,E1 25.1272,E2 412.8941} C_DIS
LIN {X 93.2545,Y 67.8501,Z 119,A 31.2478,B 24.9403,C -1.7841,E1 25.1302,E2 414.706} C_DIS
LIN {X 95.6008,Y 64.5015,Z 119,A 29.0248,B 24.9413,C -1.7701,E1 25.1338,E2 416.9511} C_DIS
LIN {X 97.413,Y 61.7338,Z 119,A 27.6037,B 24.9409,C -1.776,E1 25.1359,E2 418.3513} C_DIS
LIN {X 99.1859,Y 58.8396,Z 119,A 26.1276,B 24.9405,C -1.7812,E1 25.138,E2 419.8076} C_DIS
LIN {X 100.7519,Y 56.1158,Z 119,A 24.5027,B 24.941,C -1.774,E1 25.1402,E2 421.4411} C_DIS
LIN {X 102.5848,Y 52.6909,Z 119,A 22.0792,B 24.9429,C -1.7458,E1 25.1434,E2 423.9181} C_DIS
LIN {X 104.3384,Y 49.1292,Z 119,A 20.7086,B 24.9414,C -1.768,E1 25.145,E2 425.2291} C_DIS
LIN {X 105.5532,Y 46.4608,Z 119,A 19.0953,B 24.9422,C -1.7565,E1 25.1468,E2 426.8608} C_DIS
LIN {X 107.1856,Y 42.5599,Z 119,A 16.853,B 24.943,C -1.7438,E1 25.1492,E2 429.1206} C_DIS
LIN {X 108.8384,Y 38.133,Z 119,A 14.7538,B 24.9427,C -1.7483,E1 25.1512,E2 431.1974} C_DIS
LIN {X 110.0409,Y 34.5116,Z 119,A 12.9117,B 24.9429,C -1.745,E1 25.1528,E2 433.0367} C_DIS
LIN {X 110.764,Y 32.121,Z 119,A 11.4961,B 24.9437,C -1.7331,E1 25.1539,E2 434.4725} C_DIS
LIN {X 111.8747,Y 28.008,Z 119,A 9.2262,B 24.9446,C -1.7194,E1 25.1555,E2 436.7617} C_DIS
LIN {X 113.1966,Y 22.0572,Z 119,A 6.7848,B 24.9434,C -1.7373,E1 25.1569,E2 439.1465} C_DIS
LIN {X 113.9042,Y 18.0539,Z 119,A 4.5004,B 24.9447,C -1.7185,E1 25.158,E2 441.4619} C_DIS
LIN {X 114.3752,Y 14.773,Z 119,A 2.8968,B 24.9449,C -1.7152,E1 25.1586,E2 443.0637} C_DIS
LIN {X 114.7797,Y 11.2218,Z 119,A 0.9324,B 24.9458,C -1.7007,E1 25.1592,E2 445.0509} C_DIS
LIN {X 115.1455,Y 6.4361,Z 119,A -1.2328,B 24.9456,C -1.7032,E1 25.1596,E2 447.1971} C_DIS
LIN {X 115.2935,Y 2.7858,Z 119,A -3.1433,B 24.9463,C -1.6928,E1 25.1598,E2 449.1207} C_DIS
LIN {X 115.3116,Y -1.8025,Z 119,A -5.5179,B 24.947,C -1.681,E1 25.1598,E2 451.5092} C_DIS
LIN {X 115.1772,Y -5.8633,Z 119,A -7.3034,B 24.9468,C -1.6853,E1 25.1595,E2 453.2739} C_DIS
LIN {X 114.9677,Y -9.075,Z 119,A -8.844,B 24.9469,C -1.6828,E1 25.1592,E2 454.8111} C_DIS
LIN {X 114.5053,Y -13.7319,Z 119,A -11.1592,B 24.9474,C -1.6757,E1 25.1585,E2 457.1294} C_DIS
LIN {X 113.8195,Y -18.5807,Z 119,A -13.6938,B 24.9482,C -1.663,E1 25.1575,E2 459.6791} C_DIS
LIN {X 113.2724,Y -21.6634,Z 119,A -15.0888,B 24.948,C -1.6655,E1 25.1568,E2 461.06} C_DIS
LIN {X 112.5792,Y -25.021,Z 119,A -16.8108,B 24.9484,C -1.6591,E1 25.1558,E2 462.7871} C_DIS
LIN {X 111.4751,Y -29.5551,Z 119,A -19.262,B 24.9493,C -1.6454,E1 25.1541,E2 465.2564} C_DIS
LIN {X 110.4849,Y -33.0617,Z 119,A -21.0435,B 24.9495,C -1.641,E1 25.1527,E2 467.0382} C_DIS
LIN {X 109.5169,Y -36.1443,Z 119,A -22.4997,B 24.9495,C -1.6429,E1 25.1515,E2 468.4817} C_DIS
LIN {X 108.4731,Y -39.1617,Z 119,A -24.121,B 24.9498,C -1.6362,E1 25.15,E2 470.1095} C_DIS
LIN {X 107.4556,Y -41.8725,Z 119,A -25.6009,B 24.9502,C -1.6298,E1 25.1485,E2 471.5963} C_DIS
LIN {X 105.7636,Y -45.9782,Z 119,A -27.8367,B 24.9507,C -1.6216,E1 25.1461,E2 473.8392} C_DIS
LIN {X 104.5443,Y -48.6868,Z 119,A -29.8542,B 24.9525,C -1.5919,E1 25.1436,E2 475.9158} C_DIS
LIN {X 102.5659,Y -52.7279,Z 119,A -31.4607,B 24.9512,C -1.6144,E1 25.1417,E2 477.4607} C_DIS
LIN {X 99.6069,Y -58.1274,Z 119,A -34.6808,B 24.9522,C -1.5978,E1 25.1372,E2 480.7031} C_DIS
LIN {X 96.6806,Y -62.8746,Z 119,A -37.2008,B 24.9519,C -1.6015,E1 25.1335,E2 483.2016} C_DIS
LIN {X 94.9403,Y -65.4709,Z 119,A -38.8468,B 24.9525,C -1.5928,E1 25.1309,E2 484.86} C_DIS
LIN {X 92.8692,Y -68.3764,Z 119,A -40.6632,B 24.9529,C -1.5859,E1 25.1279,E2 486.6841} C_DIS
LIN {X 90.5969,Y -71.3593,Z 119,A -42.3999,B 24.9529,C -1.5867,E1 25.125,E2 488.4106} C_DIS
LIN {X 88.3383,Y -74.1389,Z 119,A -44.2745,B 24.9534,C -1.5775,E1 25.1216,E2 490.2982} C_DIS
LIN {X 85.8461,Y -77.009,Z 119,A -46.0456,B 24.9534,C -1.5781,E1 25.1184,E2 492.06} C_DIS
LIN {X 83.3166,Y -79.7397,Z 119,A -47.8465,B 24.9534,C -1.5757,E1 25.1149,E2 493.8589} C_DIS
LIN {X 81.1062,Y -81.986,Z 119,A -49.3816,B 24.9536,C -1.5732,E1 25.1119,E2 495.3932} C_DIS
LIN {X 78.9587,Y -84.0562,Z 119,A -50.9147,B 24.954,C -1.5673,E1 25.1088,E2 496.934} C_DIS
LIN {X 76.0596,Y -86.6886,Z 119,A -52.8579,B 24.9542,C -1.5628,E1 25.1047,E2 498.8799} C_DIS
LIN {X 73.6808,Y -88.719,Z 119,A -54.4261,B 24.9545,C -1.5586,E1 25.1014,E2 500.452} C_DIS
LIN {X 70.5804,Y -91.2051,Z 119,A -56.3361,B 24.9545,C -1.5572,E1 25.0972,E2 502.3582} C_DIS
LIN {X 67.8846,Y -93.2292,Z 119,A -58.0836,B 24.955,C -1.5503,E1 25.0933,E2 504.1157} C_DIS
LIN {X 64.8666,Y -95.3536,Z 119,A -59.9871,B 24.9554,C -1.5434,E1 25.0889,E2 506.0291} C_DIS
LIN {X 61.2267,Y -97.7304,Z 119,A -61.8627,B 24.9549,C -1.5522,E1 25.0845,E2 507.8779} C_DIS
LIN {X 59.2644,Y -98.9348,Z 119,A -63.2518,B 24.9556,C -1.5388,E1 25.0811,E2 509.2943} C_DIS
LIN {X 56.0933,Y -100.7645,Z 119,A -64.8556,B 24.9553,C -1.5453,E1 25.0773,E2 510.8778} C_DIS
LIN {X 53.5675,Y -102.1297,Z 119,A -66.9995,B 24.9573,C -1.5103,E1 25.0718,E2 513.0984} C_DIS
LIN {X 49.5776,Y -104.1256,Z 119,A -68.6813,B 24.9561,C -1.5309,E1 25.0677,E2 514.7273} C_DIS
LIN {X 42.0203,Y -107.3976,Z 119,A -72.627,B 24.9561,C -1.5314,E1 25.0576,E2 518.6625} C_DIS
LIN {X 38.7362,Y -108.6267,Z 119,A -74.4487,B 24.9564,C -1.5254,E1 25.0528,E2 520.4944} C_DIS
LIN {X 35.795,Y -109.63,Z 119,A -76.0115,B 24.9566,C -1.5227,E1 25.0486,E2 522.0607} C_DIS
LIN {X 32.0773,Y -110.7763,Z 119,A -78.0284,B 24.9569,C -1.5166,E1 25.0432,E2 524.0883} C_DIS
LIN {X 27.9618,Y -111.886,Z 119,A -80.0172,B 24.9567,C -1.5202,E1 25.0379,E2 526.0657} C_DIS
LIN {X 22.505,Y -113.1093,Z 119,A -82.838,B 24.957,C -1.5158,E1 25.0302,E2 528.8933} C_DIS
LIN {X 16.1581,Y -114.1877,Z 119,A -85.9603,B 24.9569,C -1.5168,E1 25.0216,E2 532.0102} C_DIS
LIN {X 12.3233,Y -114.6654,Z 119,A -88.3125,B 24.958,C -1.4965,E1 25.0149,E2 534.4086} C_DIS
LIN {X 8.648,Y -115.0018,Z 119,A -89.644,B 24.9568,C -1.5177,E1 25.0113,E2 535.6892} C_DIS
LIN {X 4.1279,Y -115.2529,Z 119,A -92.0407,B 24.9573,C -1.5103,E1 25.0046,E2 538.1027} C_DIS
LIN {X 0.7998,Y -115.3213,Z 119,A -92.951,B 24.9554,C -1.5428,E1 25.0023,E2 538.9358} C_DIS
Enddeposition()
LIN {X 0.7998,Y -115.3213,Z 119,A -92.951,B 24.9554,C -1.5428,E1 25.0023,E2 538.9358} C_DIS
Startdeposition()
$VEL.CP = VEL_PRINT
LIN {X 1.2208,Y -114.4284,Z 119,A -92.558,B 24.954,C -1.5663,E1 25.0035,E2 538.487} C_DIS
LIN {X 8.1476,Y -114.1441,Z 119,A -89.3615,B 24.9547,C -1.5555,E1 25.0124,E2 535.3174} C_DIS
LIN {X 13.9622,Y -113.5806,Z 119,A -86.2204,B 24.954,C -1.5667,E1 25.0212,E2 532.1518} C_DIS
LIN {X 19.0186,Y -112.8423,Z 119,A -83.6714,B 24.954,C -1.5681,E1 25.0282,E2 529.6018} C_DIS
LIN {X 21.8975,Y -112.3194,Z 119,A -81.6933,B 24.9525,C -1.5925,E1 25.0338,E2 527.5683} C_DIS
LIN {X 25.9756,Y -111.4468,Z 119,A -80.2689,B 24.9541,C -1.5645,E1 25.0375,E2 526.2121} C_DIS
LIN {X 28.7389,Y -110.7665,Z 119,A -78.8348,B 24.9541,C -1.5664,E1 25.0414,E2 524.7758} C_DIS
LIN {X 32.362,Y -109.7625,Z 119,A -76.9032,B 24.9538,C -1.5707,E1 25.0466,E2 522.8371} C_DIS
LIN {X 35.406,Y -108.8188,Z 119,A -75.3403,B 24.9538,C -1.5711,E1 25.0507,E2 521.2762} C_DIS
LIN {X 38.3776,Y -107.8077,Z 119,A -73.4225,B 24.9527,C -1.5889,E1 25.0559,E2 519.3202} C_DIS
LIN {X 42.0943,Y -106.4106,Z 119,A -70.8307,B 24.9509,C -1.6194,E1 25.0628,E2 516.6619} C_DIS
LIN {X 47.3237,Y -104.1905,Z 119,A -68.9557,B 24.9533,C -1.5792,E1 25.0673,E2 514.8867} C_DIS
LIN {X 50.1136,Y -102.8789,Z 119,A -66.8569,B 24.9516,C -1.6072,E1 25.0727,E2 512.7273} C_DIS
LIN {X 53.5151,Y -101.1496,Z 119,A -65.2561,B 24.9523,C -1.5962,E1 25.0766,E2 511.1569} C_DIS
LIN {X 57.0533,Y -99.1968,Z 119,A -63.4604,B 24.9527,C -1.5894,E1 25.0809,E2 509.3827} C_DIS
LIN {X 60.2629,Y -97.2812,Z 119,A -61.5746,B 24.9524,C -1.5936,E1 25.0854,E2 507.4929} C_DIS
LIN {X 63.6102,Y -95.1276,Z 119,A -59.6708,B 24.9524,C -1.5934,E1 25.0899,E2 505.5957} C_DIS
LIN {X 67.0304,Y -92.7496,Z 119,A -57.3809,B 24.9516,C -1.6071,E1 25.0951,E2 503.2814} C_DIS
LIN {X 69.9607,Y -90.5571,Z 119,A -55.6664,B 24.9516,C -1.6057,E1 25.0989,E2 501.5766} C_DIS
LIN {X 72.9611,Y -88.1578,Z 119,A -53.775,B 24.9516,C -1.6085,E1 25.103,E2 499.6858} C_DIS
LIN {X 75.4493,Y -86.0379,Z 119,A -52.1898,B 24.9514,C -1.6098,E1 25.1064,E2 498.1035} C_DIS
LIN {X 77.6059,Y -84.0981,Z 119,A -50.6646,B 24.951,C -1.6167,E1 25.1095,E2 496.5683} C_DIS
LIN {X 80.3775,Y -81.4527,Z 119,A -48.8091,B 24.951,C -1.6184,E1 25.1132,E2 494.7165} C_DIS
LIN {X 82.5056,Y -79.2964,Z 119,A -47.294,B 24.9507,C -1.6221,E1 25.1162,E2 493.1991} C_DIS
LIN {X 85.1142,Y -76.4898,Z 119,A -45.3324,B 24.9503,C -1.629,E1 25.1199,E2 491.2298} C_DIS
LIN {X 87.7016,Y -73.5101,Z 119,A -43.3619,B 24.95,C -1.6339,E1 25.1235,E2 489.2567} C_DIS
LIN {X 89.8481,Y -70.869,Z 119,A -41.7241,B 24.9499,C -1.6354,E1 25.1263,E2 487.623} C_DIS
LIN {X 91.7447,Y -68.3971,Z 119,A -40.0675,B 24.9493,C -1.6442,E1 25.1291,E2 485.9536} C_DIS
LIN {X 93.7792,Y -65.5793,Z 119,A -38.3649,B 24.9491,C -1.6473,E1 25.1319,E2 484.252} C_DIS
LIN {X 95.8979,Y -62.4427,Z 119,A -35.9744,B 24.9474,C -1.6761,E1 25.1356,E2 481.8056} C_DIS
LIN {X 98.1473,Y -58.8438,Z 119,A -34.5199,B 24.9489,C -1.6506,E1 25.1377,E2 480.4187} C_DIS
LIN {X 99.5854,Y -56.373,Z 119,A -32.8093,B 24.9479,C -1.668,E1 25.1401,E2 478.6759} C_DIS
LIN {X 101.8212,Y -52.2258,Z 119,A -30.5294,B 24.9477,C -1.6713,E1 25.143,E2 476.4002} C_DIS
LIN {X 103.9456,Y -47.8603,Z 119,A -28.3047,B 24.9478,C -1.6689,E1 25.1457,E2 474.1931} C_DIS
LIN {X 106.1595,Y -42.7252,Z 119,A -25.5235,B 24.9473,C -1.6767,E1 25.1487,E2 471.4088} C_DIS
LIN {X 107.3767,Y -39.5657,Z 119,A -23.4309,B 24.9458,C -1.7008,E1 25.1508,E2 469.2711} C_DIS
LIN {X 108.4558,Y -36.5022,Z 119,A -22.203,B 24.9467,C -1.6871,E1 25.1518,E2 468.0824} C_DIS
LIN {X 109.4044,Y -33.5539,Z 119,A -20.56,B 24.9461,C -1.6963,E1 25.1532,E2 466.4269} C_DIS
LIN {X 110.4899,Y -29.7837,Z 119,A -18.664,B 24.9459,C -1.6994,E1 25.1546,E2 464.5345} C_DIS
LIN {X 112.1162,Y -22.9137,Z 119,A -15.2947,B 24.9457,C -1.7029,E1 25.1567,E2 461.1765} C_DIS
LIN {X 112.6623,Y -20.0579,Z 119,A -12.8849,B 24.9424,C -1.753,E1 25.158,E2 458.6628} C_DIS
LIN {X 113.4865,Y -14.6927,Z 119,A -11.3542,B 24.9455,C -1.7054,E1 25.1585,E2 457.2532} C_DIS
LIN {X 114.0614,Y -9.2234,Z 119,A -8.3625,B 24.9442,C -1.7256,E1 25.1594,E2 454.2317} C_DIS
LIN {X 114.2653,Y -6.2062,Z 119,A -6.5622,B 24.943,C -1.7441,E1 25.1596,E2 452.3986} C_DIS
LIN {X 114.4192,Y -1.838,Z 119,A -4.7348,B 24.9436,C -1.7341,E1 25.1598,E2 450.6055} C_DIS
LIN {X 114.4238,Y 1.5883,Z 119,A -2.8468,B 24.9427,C -1.7478,E1 25.1598,E2 448.6964} C_DIS
LIN {X 114.2977,Y 5.6193,Z 119,A -0.4787,B 24.9412,C -1.7709,E1 25.1595,E2 446.288} C_DIS
LIN {X 114.0736,Y 9.0716,Z 119,A 1.2373,B 24.9409,C -1.7758,E1 25.1591,E2 444.5707} C_DIS
LIN {X 113.7255,Y 12.7253,Z 119,A 2.5226,B 24.9422,C -1.7555,E1 25.1587,E2 443.3407} C_DIS
LIN {X 113.1557,Y 17.0603,Z 119,A 5.5301,B 24.9392,C -1.8013,E1 25.1575,E2 440.2431} C_DIS
LIN {X 112.3305,Y 21.84,Z 119,A 7.9752,B 24.9386,C -1.8097,E1 25.1561,E2 437.7924} C_DIS
LIN {X 111.2595,Y 26.768,Z 119,A 9.517,B 24.9412,C -1.7711,E1 25.1553,E2 436.3504} C_DIS
LIN {X 109.9108,Y 31.8615,Z 119,A 12.2895,B 24.9402,C -1.7855,E1 25.1532,E2 433.5599} C_DIS
LIN {X 108.9022,Y 35.1482,Z 119,A 14.0532,B 24.9398,C -1.7928,E1 25.1517,E2 431.7891} C_DIS
LIN {X 107.8749,Y 38.1861,Z 119,A 15.7592,B 24.9391,C -1.8023,E1 25.1501,E2 430.0703} C_DIS
LIN {X 105.8002,Y 43.6078,Z 119,A 18.4679,B 24.9391,C -1.8016,E1 25.1474,E2 427.3782} C_DIS
LIN {X 104.4604,Y 46.7247,Z 119,A 21.2085,B 24.9355,C -1.8555,E1 25.1442,E2 424.5254} C_DIS
LIN {X 101.8721,Y 52.1263,Z 119,A 23.1296,B 24.9384,C -1.8133,E1 25.1419,E2 422.714} C_DIS
LIN {X 100.5268,Y 54.6758,Z 119,A 24.6809,B 24.9378,C -1.8224,E1 25.1398,E2 421.1496} C_DIS
LIN {X 98.5003,Y 58.2475,Z 119,A 26.6513,B 24.9376,C -1.824,E1 25.1371,E2 419.1856} C_DIS
LIN {X 96.7622,Y 61.0938,Z 119,A 28.6641,B 24.9362,C -1.8443,E1 25.134,E2 417.135} C_DIS
LIN {X 94.0799,Y 65.1467,Z 119,A 30.8556,B 24.9366,C -1.8394,E1 25.1306,E2 414.9659} C_DIS
LIN {X 91.4834,Y 68.745,Z 119,A 32.9145,B 24.9367,C -1.8374,E1 25.1273,E2 412.9216} C_DIS
LIN {X 89.6701,Y 71.0941,Z 119,A 35.1691,B 24.934,C -1.8766,E1 25.1232,E2 410.585} C_DIS
LIN {X 86.5647,Y 74.8462,Z 119,A 36.7673,B 24.9363,C -1.8434,E1 25.1205,E2 409.0724} C_DIS
LIN {X 83.3168,Y 78.4436,Z 119,A 39.2785,B 24.9357,C -1.8528,E1 25.1157,E2 406.5502} C_DIS
LIN {X 81.3938,Y 80.4371,Z 119,A 40.6587,B 24.9355,C -1.8555,E1 25.113,E2 405.1695} C_DIS
LIN {X 79.0534,Y 82.7398,Z 119,A 43.2037,B 24.9323,C -1.9004,E1 25.1077,E2 402.5289} C_DIS
LIN {X 74.9245,Y 86.4963,Z 119,A 45.0496,B 24.935,C -1.8624,E1 25.104,E2 400.7801} C_DIS
LIN {X 70.6711,Y 90.0045,Z 119,A 47.6569,B 24.9351,C -1.8607,E1 25.0984,E2 398.1869} C_DIS
LIN {X 68.716,Y 91.5051,Z 119,A 49.1146,B 24.9342,C -1.873,E1 25.0951,E2 396.7053} C_DIS
LIN {X 65.0418,Y 94.1528,Z 119,A 51.2985,B 24.9342,C -1.8731,E1 25.0902,E2 394.5286} C_DIS
LIN {X 62.3523,Y 95.9563,Z 119,A 52.8659,B 24.9342,C -1.8733,E1 25.0865,E2 392.966} C_DIS
LIN {X 59.6647,Y 97.6487,Z 119,A 54.5874,B 24.9336,C -1.8817,E1 25.0824,E2 391.2302} C_DIS
LIN {X 54.2717,Y 100.746,Z 119,A 57.5488,B 24.9338,C -1.8793,E1 25.0752,E2 388.2833} C_DIS
LIN {X 51.5711,Y 102.1558,Z 119,A 59.27,B 24.933,C -1.89,E1 25.0709,E2 386.5414} C_DIS
LIN {X 45.3474,Y 105.066,Z 119,A 62.462,B 24.9335,C -1.883,E1 25.0629,E2 383.3741} C_DIS
LIN {X 40.8471,Y 106.8958,Z 119,A 64.8228,B 24.9335,C -1.8823,E1 25.0568,E2 381.0204} C_DIS
LIN {X 37.2648,Y 108.1982,Z 119,A 66.8653,B 24.933,C -1.8899,E1 25.0514,E2 378.964} C_DIS
LIN {X 34.4618,Y 109.1229,Z 119,A 68.4884,B 24.9325,C -1.8975,E1 25.047,E2 377.3259} C_DIS
LIN {X 30.9103,Y 110.1804,Z 119,A 70.1797,B 24.9329,C -1.8916,E1 25.0425,E2 375.6514} C_DIS
LIN {X 27.7002,Y 111.0321,Z 119,A 71.9753,B 24.9324,C -1.8985,E1 25.0376,E2 373.8424} C_DIS
LIN {X 23.082,Y 112.0817,Z 119,A 74.1794,B 24.9329,C -1.8924,E1 25.0317,E2 371.6556} C_DIS
LIN {X 17.5888,Y 113.0739,Z 119,A 76.7503,B 24.9335,C -1.8836,E1 25.0247,E2 369.1082} C_DIS
LIN {X 11.9358,Y 113.8095,Z 119,A 80.5972,B 24.9304,C -1.9274,E1 25.0137,E2 365.1604} C_DIS
LIN {X 7.3313,Y 114.1993,Z 119,A 82.2373,B 24.9325,C -1.8981,E1 25.0093,E2 363.5905} C_DIS
LIN {X 0.4251,Y 114.4332,Z 119,A 85.4362,B 24.9333,C -1.8865,E1 25.0005,E2 360.4199} C_DIS
LIN {X -4.3448,Y 114.3526,Z 119,A 88.1006,B 24.9325,C -1.8976,E1 24.993,E2 357.7289} C_DIS
LIN {X -12.4134,Y 113.7595,Z 119,A 93.1241,B 24.9296,C -1.9375,E1 24.9787,E2 352.6081} C_DIS
LIN {X -18.3051,Y 112.9616,Z 119,A 95.0188,B 24.9331,C -1.889,E1 24.9738,E2 350.8269} C_DIS
LIN {X -26.8052,Y 111.2504,Z 119,A 99.2567,B 24.9337,C -1.8809,E1 24.9623,E2 346.6033} C_DIS
LIN {X -30.483,Y 110.3009,Z 119,A 101.514,B 24.9328,C -1.8939,E1 24.9561,E2 344.3118} C_DIS
LIN {X -35.2958,Y 108.8544,Z 119,A 103.5038,B 24.9345,C -1.869,E1 24.9509,E2 342.3778} C_DIS
LIN {X -37.3887,Y 108.1547,Z 119,A 105.1072,B 24.9331,C -1.8884,E1 24.9465,E2 340.7251} C_DIS
LIN {X -43.5381,Y 105.8283,Z 119,A 108.4151,B 24.9334,C -1.8846,E1 24.938,E2 337.4192} C_DIS
LIN {X -49.8417,Y 103.0096,Z 119,A 111.756,B 24.9341,C -1.8744,E1 24.9295,E2 334.0943} C_DIS
LIN {X -53.0998,Y 101.3684,Z 119,A 114.2237,B 24.9325,C -1.8981,E1 24.9232,E2 331.5635} C_DIS
LIN {X -56.8489,Y 99.3142,Z 119,A 116.242,B 24.9331,C -1.8892,E1 24.9184,E2 329.5605} C_DIS
LIN {X -60.1122,Y 97.3754,Z 119,A 117.5819,B 24.935,C -1.8624,E1 24.9153,E2 328.2802} C_DIS
LIN {X -65.3398,Y 93.9456,Z 119,A 121.1457,B 24.9342,C -1.8741,E1 24.907,E2 324.6768} C_DIS
LIN {X -68.6913,Y 91.5236,Z 119,A 122.843,B 24.9355,C -1.8544,E1 24.9032,E2 323.0203} C_DIS
LIN {X -71.1178,Y 89.6514,Z 119,A 124.4424,B 24.9355,C -1.8537,E1 24.8997,E2 321.4166} C_DIS
LIN {X -75.1872,Y 86.2669,Z 119,A 127.4548,B 24.935,C -1.8626,E1 24.8932,E2 318.3714} C_DIS
LIN {X -78.6857,Y 83.089,Z 119,A 129.573,B 24.9361,C -1.8468,E1 24.889,E2 316.2821} C_DIS
LIN {X -81.4388,Y 80.3915,Z 119,A 131.8374,B 24.9354,C -1.8558,E1 24.8844,E2 313.9867} C_DIS
LIN {X -83.8795,Y 77.8435,Z 119,A 133.7613,B 24.9354,C -1.8578,E1 24.8808,E2 312.0497} C_DIS
LIN {X -86.6266,Y 74.7753,Z 119,A 135.4068,B 24.9369,C -1.8354,E1 24.8778,E2 310.4499} C_DIS
LIN {X -89.1093,Y 71.7963,Z 119,A 137.978,B 24.9354,C -1.856,E1 24.8732,E2 307.8177} C_DIS
LIN {X -92.1165,Y 67.8952,Z 119,A 139.9147,B 24.9374,C -1.8277,E1 24.8701,E2 305.9393} C_DIS
LIN {X -95.3289,Y 63.3057,Z 119,A 142.3294,B 24.939,C -1.8041,E1 24.8663,E2 303.5688} C_DIS
LIN {X -96.8433,Y 60.964,Z 119,A 144.6439,B 24.9367,C -1.8373,E1 24.8628,E2 301.1634} C_DIS
LIN {X -99.2663,Y 56.9322,Z 119,A 146.2344,B 24.9393,C -1.7994,E1 24.8606,E2 299.655} C_DIS
LIN {X -101.5339,Y 52.7855,Z 119,A 148.7127,B 24.9395,C -1.7969,E1 24.8573,E2 297.1696} C_DIS
LIN {X -103.6884,Y 48.4129,Z 119,A 150.9611,B 24.9405,C -1.7818,E1 24.8546,E2 294.9449} C_DIS
LIN {X -106.5568,Y 41.7221,Z 119,A 154.7454,B 24.9409,C -1.7761,E1 24.8505,E2 291.1532} C_DIS
LIN {X -108.902,Y 35.1488,Z 119,A 158.3417,B 24.9413,C -1.7691,E1 24.8472,E2 287.5531} C_DIS
LIN {X -109.7934,Y 32.2578,Z 119,A 159.9743,B 24.9413,C -1.7691,E1 24.8459,E2 285.9113} C_DIS
LIN {X -111.6858,Y 24.9335,Z 119,A 163.5549,B 24.9427,C -1.7486,E1 24.8435,E2 282.3586} C_DIS
LIN {X -112.4401,Y 21.2702,Z 119,A 165.6369,B 24.9425,C -1.7509,E1 24.8423,E2 280.2588} C_DIS
LIN {X -113.3515,Y 15.7056,Z 119,A 168.3248,B 24.9435,C -1.7363,E1 24.8412,E2 277.5897} C_DIS
LIN {X -113.9305,Y 10.7219,Z 119,A 170.6522,B 24.9445,C -1.7207,E1 24.8405,E2 275.2854} C_DIS
LIN {X -114.1546,Y 7.9926,Z 119,A 172.3569,B 24.9439,C -1.7296,E1 24.8401,E2 273.5494} C_DIS
LIN {X -114.4001,Y 2.8504,Z 119,A 175.4894,B 24.943,C -1.7435,E1 24.8398,E2 270.3648} C_DIS
LIN {X -114.4279,Y -1.3145,Z 119,A 176.9497,B 24.9451,C -1.7116,E1 24.8398,E2 268.9719} C_DIS
LIN {X -114.3438,Y -4.5497,Z 119,A 179.2864,B 24.9436,C -1.7352,E1 24.8401,E2 266.5647} C_DIS
LIN {X -114.0812,Y -8.9765,Z 119,A -178.6005,B 24.9443,C -1.7237,E1 24.8405,E2 264.4664} C_DIS
LIN {X -113.7032,Y -12.9152,Z 119,A -177.3199,B 24.9465,C -1.6891,E1 24.8409,E2 263.2607} C_DIS
LIN {X -113.3675,Y -15.593,Z 119,A -175.1751,B 24.9448,C -1.7168,E1 24.8417,E2 261.037} C_DIS
LIN {X -112.7146,Y -19.7671,Z 119,A -173.7843,B 24.9471,C -1.6808,E1 24.8424,E2 259.7238} C_DIS
LIN {X -111.9692,Y -23.6297,Z 119,A -171.5172,B 24.9467,C -1.6866,E1 24.8436,E2 257.4296} C_DIS
LIN {X -111.0511,Y -27.6223,Z 119,A -169.6322,B 24.9475,C -1.6735,E1 24.8448,E2 255.5647} C_DIS
LIN {X -110.111,Y -31.1551,Z 119,A -167.7648,B 24.9478,C -1.6694,E1 24.8462,E2 253.6962} C_DIS
LIN {X -109.1245,Y -34.4566,Z 119,A -165.7185,B 24.9473,C -1.6771,E1 24.8479,E2 251.6197} C_DIS
LIN {X -107.2908,Y -39.7979,Z 119,A -162.9366,B 24.9479,C -1.6668,E1 24.8505,E2 248.8467} C_DIS
LIN {X -105.5431,Y -44.2243,Z 119,A -160.4845,B 24.9482,C -1.6626,E1 24.8531,E2 246.3907} C_DIS
LIN {X -103.76,Y -48.2591,Z 119,A -158.5471,B 24.9493,C -1.6453,E1 24.8553,E2 244.4842} C_DIS
LIN {X -102.2651,Y -51.3544,Z 119,A -156.6808,B 24.9493,C -1.6463,E1 24.8576,E2 242.6054} C_DIS
LIN {X -99.174,Y -57.0929,Z 119,A -153.9431,B 24.9511,C -1.6159,E1 24.8612,E2 239.9256} C_DIS
LIN {X -95.2729,Y -63.3907,Z 119,A -149.9902,B 24.9511,C -1.6159,E1 24.8671,E2 235.9525} C_DIS
LIN {X -92.831,Y -66.9163,Z 119,A -146.9023,B 24.949,C -1.6493,E1 24.8722,E2 232.77} C_DIS
LIN {X -89.9357,Y -70.7581,Z 119,A -145.4746,B 24.9519,C -1.6029,E1 24.8745,E2 231.4461} C_DIS
LIN {X -87.4729,Y -73.7827,Z 119,A -143.1577,B 24.9512,C -1.6132,E1 24.8787,E2 229.0939} C_DIS
LIN {X -85.066,Y -76.5436,Z 119,A -141.5582,B 24.9521,C -1.5993,E1 24.8816,E2 227.5202} C_DIS
LIN {X -83.2501,Y -78.5145,Z 119,A -140.0462,B 24.9518,C -1.6034,E1 24.8845,E2 225.992} C_DIS
LIN {X -78.5358,Y -83.23,Z 119,A -136.7253,B 24.9523,C -1.5955,E1 24.8911,E2 222.6758} C_DIS
LIN {X -76.212,Y -85.3629,Z 119,A -135.1351,B 24.9525,C -1.5928,E1 24.8944,E2 221.0858} C_DIS
LIN {X -73.1536,Y -87.9978,Z 119,A -133.1967,B 24.9529,C -1.5854,E1 24.8985,E2 219.1574} C_DIS
LIN {X -70.9185,Y -89.8089,Z 119,A -131.6129,B 24.9527,C -1.5888,E1 24.902,E2 217.5597} C_DIS
LIN {X -67.8394,Y -92.1573,Z 119,A -129.6863,B 24.9529,C -1.5848,E1 24.9062,E2 215.6356} C_DIS
LIN {X -64.0398,Y -94.8367,Z 119,A -127.4677,B 24.9534,C -1.5763,E1 24.9113,E2 213.4296} C_DIS
LIN {X -61.5978,Y -96.4409,Z 119,A -125.2603,B 24.9517,C -1.6056,E1 24.9167,E2 211.1456} C_DIS
LIN {X -57.7853,Y -98.7734,Z 119,A -123.6778,B 24.9536,C -1.5744,E1 24.9203,E2 209.6324} C_DIS
LIN {X -54.6495,Y -100.5411,Z 119,A -121.8658,B 24.9536,C -1.5723,E1 24.9247,E2 207.8201} C_DIS
LIN {X -48.3463,Y -103.7194,Z 119,A -118.3076,B 24.9539,C -1.5689,E1 24.9337,E2 204.2607} C_DIS
LIN {X -43.7456,Y -105.7441,Z 119,A -115.8503,B 24.9542,C -1.5636,E1 24.9399,E2 201.8103} C_DIS
LIN {X -39.7373,Y -107.3142,Z 119,A -113.7321,B 24.9544,C -1.5599,E1 24.9454,E2 199.6962} C_DIS
LIN {X -37.1077,Y -108.2517,Z 119,A -112.1265,B 24.954,C -1.5677,E1 24.9497,E2 198.0692} C_DIS
LIN {X -33.7571,Y -109.3414,Z 119,A -110.4887,B 24.9544,C -1.5609,E1 24.9541,E2 196.4445} C_DIS
LIN {X -30.7364,Y -110.2296,Z 119,A -108.8828,B 24.9544,C -1.5611,E1 24.9584,E2 194.8355} C_DIS
LIN {X -26.12,Y -111.4134,Z 119,A -106.6816,B 24.9549,C -1.5517,E1 24.9643,E2 192.6534} C_DIS
LIN {X -22.5489,Y -112.1911,Z 119,A -104.6905,B 24.9545,C -1.5579,E1 24.9698,E2 190.6453} C_DIS
LIN {X -19.6487,Y -112.7359,Z 119,A -102.5945,B 24.953,C -1.5845,E1 24.9757,E2 188.4842} C_DIS
LIN {X -15.5471,Y -113.374,Z 119,A -100.6887,B 24.9534,C -1.5764,E1 24.9809,E2 186.596} C_DIS
LIN {X -12.2307,Y -113.7786,Z 119,A -99.6432,B 24.9551,C -1.5487,E1 24.9837,E2 185.6156} C_DIS
LIN {X -8.0681,Y -114.1495,Z 119,A -96.8584,B 24.9533,C -1.5791,E1 24.9916,E2 182.7575} C_DIS
LIN {X -4.3273,Y -114.3534,Z 119,A -94.8632,B 24.953,C -1.5846,E1 24.9972,E2 180.749} C_DIS
LIN {X -0.1106,Y -114.4352,Z 119,A -93.392,B 24.9546,C -1.5566,E1 25.0011,E2 179.3441} C_DIS
LIN {X -0.1106,Y -114.4352,Z 119,A -93.392,B 24.9546,C -1.5566,E1 25.0011,E2 179.3441} C_DIS
Enddeposition()
LIN {X 0.7983,Y -113.5063,Z 119,A -93.822,B 24.9559,C -1.5343,E1 24.9998,E2 179.8268} C_DIS
Startdeposition()
$VEL.CP = VEL_PRINT
LIN {X -3.3588,Y -113.4925,Z 119,A -96.5457,B 24.9575,C -1.5067,E1 24.992,E2 182.6163} C_DIS
LIN {X -8.4949,Y -113.2253,Z 119,A -98.3087,B 24.9554,C -1.5421,E1 24.9873,E2 184.296} C_DIS
LIN {X -14.5104,Y -112.6112,Z 119,A -101.754,B 24.9564,C -1.5257,E1 24.9777,E2 187.7823} C_DIS
LIN {X -17.6796,Y -112.1577,Z 119,A -103.1312,B 24.9558,C -1.5363,E1 24.9739,E2 189.1357} C_DIS
LIN {X -23.9761,Y -110.982,Z 119,A -106.2495,B 24.9554,C -1.5424,E1 24.9654,E2 192.2429} C_DIS
LIN {X -28.3493,Y -109.9461,Z 119,A -108.5349,B 24.9554,C -1.5429,E1 24.9592,E2 194.5303} C_DIS
LIN {X -31.9417,Y -108.9572,Z 119,A -110.4485,B 24.9554,C -1.5427,E1 24.954,E2 196.4475} C_DIS
LIN {X -35.3417,Y -107.9025,Z 119,A -112.2159,B 24.9553,C -1.5453,E1 24.9493,E2 198.2118} C_DIS
Enddeposition()
END
